KUKA KRL program: MyProgram_103().src

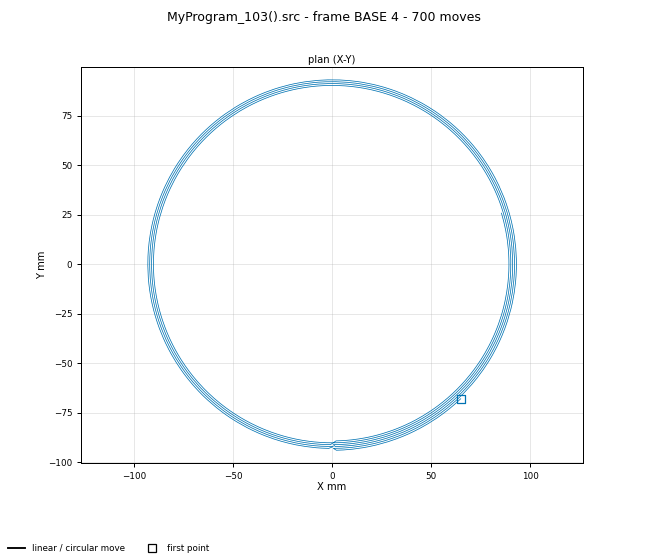
[picture p0: tool path of MyProgram_103().src in frame BASE 4, 700 of 700 moves have a stored position in this frame; points joined in program order, loops and branches not executed]
&ACCESS RVP
&REL 1
&PARAM TEMPLATE = C:\KRC\Roboter\Template\vorgabe
&PARAM EDITMASK = *
DEF MyProgram_103()
; ---- Setting reference (Base) ----
$BASE = BASE_DATA[4]

; --------------------------
; ---- Setting tool (TCP) ----
$TOOL = TOOL_DATA[3]
; --------------------------

$VEL.CP = VEL_APROX_PRINT
Startdeposition()
$VEL.CP = VEL_PRINT
LIN {X 64.9049,Y -67.9874,Z 93,A -51.9833,B 24.9346,C -1.8674,E1 25.1081,E2 497.2894} C_DIS
LIN {X 61.9537,Y -70.6859,Z 93,A -53.7014,B 24.9332,C -1.8881,E1 25.1046,E2 498.9518} C_DIS
LIN {X 59.3764,Y -72.8646,Z 93,A -56.3232,B 24.9349,C -1.863,E1 25.0988,E2 501.6231} C_DIS
LIN {X 56.5767,Y -75.0589,Z 93,A -58.0542,B 24.9341,C -1.8743,E1 25.0951,E2 503.3211} C_DIS
LIN {X 52.9467,Y -77.6626,Z 93,A -60.3598,B 24.9335,C -1.884,E1 25.0899,E2 505.5957} C_DIS
LIN {X 48.6372,Y -80.4313,Z 93,A -63.8521,B 24.9348,C -1.8645,E1 25.0815,E2 509.1227} C_DIS
LIN {X 44.582,Y -82.7481,Z 93,A -66.4916,B 24.9347,C -1.867,E1 25.0752,E2 511.7486} C_DIS
LIN {X 41.1529,Y -84.5065,Z 93,A -68.9502,B 24.9352,C -1.8591,E1 25.069,E2 514.2192} C_DIS
LIN {X 38.4528,Y -85.768,Z 93,A -70.647,B 24.9352,C -1.8607,E1 25.0647,E2 515.908} C_DIS
LIN {X 35.5579,Y -87.008,Z 93,A -72.6876,B 24.9356,C -1.8535,E1 25.0594,E2 517.9607} C_DIS
LIN {X 32.1278,Y -88.332,Z 93,A -74.8746,B 24.9356,C -1.8524,E1 25.0537,E2 520.1456} C_DIS
LIN {X 28.0038,Y -89.7249,Z 93,A -77.5473,B 24.9359,C -1.8485,E1 25.0466,E2 522.8225} C_DIS
LIN {X 22.2186,Y -91.3295,Z 93,A -81.2447,B 24.9363,C -1.8433,E1 25.0366,E2 526.5264} C_DIS
LIN {X 18.4904,Y -92.1576,Z 93,A -83.3808,B 24.936,C -1.848,E1 25.0308,E2 528.6487} C_DIS
LIN {X 15.7341,Y -92.6673,Z 93,A -85.254,B 24.9365,C -1.8409,E1 25.0256,E2 530.5368} C_DIS
LIN {X 10.3903,Y -93.4188,Z 93,A -88.3808,B 24.9362,C -1.8444,E1 25.017,E2 533.6526} C_DIS
LIN {X 5.6146,Y -93.8264,Z 93,A -91.4459,B 24.9367,C -1.838,E1 25.0084,E2 536.7313} C_DIS
LIN {X 2.1765,Y -93.9691,Z 93,A -93.605,B 24.9369,C -1.8351,E1 25.0024,E2 538.8967} C_DIS
LIN {X 2.1765,Y -93.9691,Z 93,A -93.605,B 24.9369,C -1.8351,E1 25.0024,E2 538.8967} C_DIS
Enddeposition()
LIN {X 0.6226,Y -93.0173,Z 93,A -94.0393,B 24.9345,C -1.8697,E1 25.0014,E2 539.2489} C_DIS
Startdeposition()
$VEL.CP = VEL_PRINT
LIN {X 4.8122,Y -92.9245,Z 93,A -89.9697,B 24.9307,C -1.9224,E1 25.0131,E2 535.0555} C_DIS
LIN {X 10.0586,Y -92.5039,Z 93,A -88.0458,B 24.9339,C -1.8776,E1 25.0182,E2 533.2392} C_DIS
LIN {X 16.1981,Y -91.6281,Z 93,A -83.9532,B 24.9331,C -1.8898,E1 25.0295,E2 529.1213} C_DIS
LIN {X 21.4978,Y -90.5327,Z 93,A -80.1723,B 24.9317,C -1.9088,E1 25.0399,E2 525.3004} C_DIS
LIN {X 26.3121,Y -89.2508,Z 93,A -77.5578,B 24.9326,C -1.8959,E1 25.0469,E2 522.7207} C_DIS
LIN {X 29.8863,Y -88.1184,Z 93,A -75.0169,B 24.9318,C -1.9071,E1 25.0537,E2 520.1582} C_DIS
LIN {X 33.849,Y -86.6734,Z 93,A -72.666,B 24.9322,C -1.9017,E1 25.0598,E2 517.8252} C_DIS
LIN {X 36.9367,Y -85.4035,Z 93,A -70.7563,B 24.9324,C -1.8994,E1 25.0647,E2 515.9253} C_DIS
LIN {X 40.1669,Y -83.9324,Z 93,A -67.9542,B 24.9305,C -1.9253,E1 25.0719,E2 513.0693} C_DIS
LIN {X 43.1685,Y -82.429,Z 93,A -66.412,B 24.9316,C -1.9096,E1 25.0756,E2 511.5685} C_DIS
LIN {X 45.3175,Y -81.2671,Z 93,A -64.8499,B 24.9313,C -1.9143,E1 25.0794,E2 509.9997} C_DIS
LIN {X 48.1998,Y -79.5916,Z 93,A -62.4975,B 24.9302,C -1.9291,E1 25.0851,E2 507.6197} C_DIS
LIN {X 52.1558,Y -77.057,Z 93,A -60.0101,B 24.9309,C -1.9198,E1 25.0909,E2 505.1624} C_DIS
LIN {X 55.1018,Y -74.9788,Z 93,A -57.7519,B 24.9305,C -1.9258,E1 25.096,E2 502.898} C_DIS
LIN {X 58.2189,Y -72.5845,Z 93,A -54.9321,B 24.929,C -1.9458,E1 25.1023,E2 500.0413} C_DIS
LIN {X 62.7773,Y -68.6808,Z 93,A -51.4545,B 24.929,C -1.9462,E1 25.1095,E2 496.5767} C_DIS
LIN {X 66.2243,Y -65.3632,Z 93,A -48.3301,B 24.928,C -1.96,E1 25.1157,E2 493.4329} C_DIS
LIN {X 70.519,Y -60.7043,Z 93,A -44.6552,B 24.9279,C -1.9614,E1 25.1226,E2 489.771} C_DIS
LIN {X 73.1256,Y -57.5385,Z 93,A -42.0163,B 24.9271,C -1.9724,E1 25.1272,E2 487.1185} C_DIS
LIN {X 76.178,Y -53.4329,Z 93,A -38.7924,B 24.9262,C -1.9837,E1 25.1325,E2 483.8835} C_DIS
LIN {X 79.1029,Y -48.9987,Z 93,A -35.8993,B 24.9266,C -1.9787,E1 25.1368,E2 481.0166} C_DIS
LIN {X 81.007,Y -45.7832,Z 93,A -32.8346,B 24.9239,C -2.0143,E1 25.1411,E2 477.884} C_DIS
LIN {X 83.1606,Y -41.7437,Z 93,A -30.7888,B 24.9255,C -1.9933,E1 25.1436,E2 475.8985} C_DIS
LIN {X 84.574,Y -38.8009,Z 93,A -28.9541,B 24.9255,C -1.9927,E1 25.1458,E2 474.0751} C_DIS
LIN {X 85.7557,Y -36.1106,Z 93,A -27.0884,B 24.925,C -2.0004,E1 25.1479,E2 472.2015} C_DIS
LIN {X 87.1821,Y -32.5194,Z 93,A -24.5222,B 24.9239,C -2.0147,E1 25.1504,E2 469.6157} C_DIS
LIN {X 88.5131,Y -28.6957,Z 93,A -22.2361,B 24.9239,C -2.0147,E1 25.1525,E2 467.3427} C_DIS
LIN {X 90.2836,Y -22.5193,Z 93,A -18.2449,B 24.9228,C -2.0284,E1 25.1555,E2 463.3419} C_DIS
LIN {X 90.9527,Y -19.638,Z 93,A -15.504,B 24.9197,C -2.0693,E1 25.1571,E2 460.5206} C_DIS
LIN {X 91.9008,Y -14.5732,Z 93,A -13.5998,B 24.9226,C -2.0311,E1 25.1579,E2 458.7176} C_DIS
LIN {X 92.581,Y -9.322,Z 93,A -10.0696,B 24.9211,C -2.0517,E1 25.1592,E2 455.1595} C_DIS
LIN {X 92.8553,Y -5.9982,Z 93,A -7.4727,B 24.9189,C -2.079,E1 25.1596,E2 452.5138} C_DIS
LIN {X 93.0232,Y -2.2255,Z 93,A -5.3762,B 24.919,C -2.0777,E1 25.1598,E2 450.4328} C_DIS
LIN {X 93.0129,Y 2.5845,Z 93,A -2.7784,B 24.9194,C -2.0734,E1 25.1597,E2 447.8605} C_DIS
LIN {X 92.6878,Y 8.1923,Z 93,A 0.3644,B 24.9194,C -2.0725,E1 25.1591,E2 444.7385} C_DIS
LIN {X 91.9596,Y 14.1932,Z 93,A 3.8715,B 24.9192,C -2.0762,E1 25.1579,E2 441.2436} C_DIS
LIN {X 91.3908,Y 17.4854,Z 93,A 6.6018,B 24.9167,C -2.1078,E1 25.1565,E2 438.4545} C_DIS
LIN {X 90.4897,Y 21.671,Z 93,A 9.2019,B 24.9161,C -2.1146,E1 25.1549,E2 435.8536} C_DIS
LIN {X 89.4572,Y 25.6022,Z 93,A 11.8466,B 24.9151,C -2.1275,E1 25.1529,E2 433.1936} C_DIS
LIN {X 87.9202,Y 30.4662,Z 93,A 14.5943,B 24.9155,C -2.1221,E1 25.1505,E2 430.4741} C_DIS
LIN {X 86.7849,Y 33.5653,Z 93,A 16.5323,B 24.9153,C -2.1245,E1 25.1486,E2 428.5413} C_DIS
LIN {X 84.1559,Y 39.6992,Z 93,A 20.551,B 24.9147,C -2.1328,E1 25.1442,E2 424.5249} C_DIS
LIN {X 82.2903,Y 43.4318,Z 93,A 23.7236,B 24.9123,C -2.1624,E1 25.14,E2 421.2993} C_DIS
LIN {X 80.6908,Y 46.3358,Z 93,A 25.2293,B 24.9135,C -2.1479,E1 25.138,E2 419.8355} C_DIS
LIN {X 78.7656,Y 49.5386,Z 93,A 28.4403,B 24.9102,C -2.1878,E1 25.1331,E2 416.5466} C_DIS
LIN {X 76.1381,Y 53.4898,Z 93,A 30.5308,B 24.9121,C -2.1643,E1 25.1299,E2 414.522} C_DIS
LIN {X 73.6324,Y 56.8885,Z 93,A 33.1379,B 24.9116,C -2.1709,E1 25.1255,E2 411.9117} C_DIS
LIN {X 71.2757,Y 59.8163,Z 93,A 35.2495,B 24.9118,C -2.1689,E1 25.1218,E2 409.8147} C_DIS
LIN {X 69.3808,Y 62.0025,Z 93,A 37.7076,B 24.9094,C -2.1977,E1 25.1172,E2 407.2993} C_DIS
LIN {X 66.8807,Y 64.6916,Z 93,A 39.4484,B 24.9106,C -2.1836,E1 25.1139,E2 405.5995} C_DIS
LIN {X 64.3624,Y 67.1981,Z 93,A 41.445,B 24.9108,C -2.1812,E1 25.1099,E2 403.6168} C_DIS
LIN {X 62.0278,Y 69.3582,Z 93,A 43.5422,B 24.91,C -2.1902,E1 25.1055,E2 401.5069} C_DIS
LIN {X 59.3656,Y 71.6503,Z 93,A 45.8089,B 24.9094,C -2.1981,E1 25.1007,E2 399.2303} C_DIS
LIN {X 54.7047,Y 75.2696,Z 93,A 49.3703,B 24.9091,C -2.2019,E1 25.0928,E2 395.6728} C_DIS
LIN {X 51.8989,Y 77.231,Z 93,A 51.6065,B 24.9084,C -2.2099,E1 25.0876,E2 393.425} C_DIS
LIN {X 48.6643,Y 79.3092,Z 93,A 53.9531,B 24.9081,C -2.2128,E1 25.082,E2 391.0791} C_DIS
LIN {X 45.3097,Y 81.2714,Z 93,A 56.5154,B 24.9074,C -2.2222,E1 25.0758,E2 388.5022} C_DIS
LIN {X 39.8165,Y 84.1008,Z 93,A 59.8419,B 24.9084,C -2.21,E1 25.0676,E2 385.2137} C_DIS
LIN {X 35.4139,Y 86.0465,Z 93,A 62.8769,B 24.9079,C -2.2157,E1 25.0598,E2 382.1724} C_DIS
LIN {X 31.8753,Y 87.4184,Z 93,A 65.1162,B 24.908,C -2.2145,E1 25.0539,E2 379.9407} C_DIS
LIN {X 29.3278,Y 88.3067,Z 93,A 66.9704,B 24.9073,C -2.2226,E1 25.049,E2 378.0709} C_DIS
LIN {X 25.9844,Y 89.348,Z 93,A 69.1375,B 24.9072,C -2.2246,E1 25.0432,E2 375.903} C_DIS
LIN {X 22.6331,Y 90.2555,Z 93,A 71.0724,B 24.9076,C -2.2189,E1 25.038,E2 373.9847} C_DIS
LIN {X 20.5715,Y 90.7467,Z 93,A 72.4369,B 24.9074,C -2.2216,E1 25.0343,E2 372.6155} C_DIS
LIN {X 15.3426,Y 91.7748,Z 93,A 75.7008,B 24.9074,C -2.2223,E1 25.0253,E2 369.3537} C_DIS
LIN {X 13.1156,Y 92.1194,Z 93,A 77.9313,B 24.9049,C -2.2518,E1 25.019,E2 367.0552} C_DIS
LIN {X 8.696,Y 92.6413,Z 93,A 79.8432,B 24.9073,C -2.2236,E1 25.0139,E2 365.2115} C_DIS
LIN {X 3.7542,Y 92.973,Z 93,A 82.7917,B 24.9075,C -2.2201,E1 25.0057,E2 362.2724} C_DIS
LIN {X -2.15,Y 93.0246,Z 93,A 86.4724,B 24.9075,C -2.2208,E1 24.9954,E2 358.59} C_DIS
LIN {X -7.3461,Y 92.758,Z 93,A 89.5732,B 24.9079,C -2.2162,E1 24.9868,E2 355.4994} C_DIS
LIN {X -13.9208,Y 92.0017,Z 93,A 94.8926,B 24.9046,C -2.2555,E1 24.9718,E2 350.0827} C_DIS
LIN {X -19.1569,Y 91.0562,Z 93,A 97.185,B 24.9076,C -2.2198,E1 24.9657,E2 347.8725} C_DIS
LIN {X -21.6885,Y 90.4863,Z 93,A 99.0287,B 24.907,C -2.2264,E1 24.9607,E2 346.0105} C_DIS
LIN {X -26.5562,Y 89.1784,Z 93,A 101.8447,B 24.9081,C -2.2137,E1 24.9532,E2 343.2203} C_DIS
LIN {X -29.2761,Y 88.3241,Z 93,A 103.4506,B 24.9087,C -2.2067,E1 24.9489,E2 341.6281} C_DIS
LIN {X -33.6201,Y 86.7634,Z 93,A 106.2312,B 24.9091,C -2.201,E1 24.9417,E2 338.8554} C_DIS
LIN {X -37.1622,Y 85.3052,Z 93,A 108.7868,B 24.9089,C -2.2041,E1 24.935,E2 336.2867} C_DIS
LIN {X -39.1812,Y 84.397,Z 93,A 110.6758,B 24.9076,C -2.2191,E1 24.9302,E2 334.3573} C_DIS
LIN {X -42.1939,Y 82.932,Z 93,A 112.5588,B 24.9084,C -2.2099,E1 24.9255,E2 332.4911} C_DIS
LIN {X -46.113,Y 80.8188,Z 93,A 114.9541,B 24.9097,C -2.1939,E1 24.9197,E2 330.1269} C_DIS
LIN {X -48.8364,Y 79.2042,Z 93,A 116.9522,B 24.9099,C -2.1919,E1 24.915,E2 328.1274} C_DIS
LIN {X -54.2253,Y 75.6153,Z 93,A 120.858,B 24.9107,C -2.1815,E1 24.906,E2 324.2333} C_DIS
LIN {X -55.8386,Y 74.4316,Z 93,A 122.2481,B 24.9105,C -2.184,E1 24.9028,E2 322.8324} C_DIS
LIN {X -58.7964,Y 72.1184,Z 93,A 124.6083,B 24.9108,C -2.1805,E1 24.8977,E2 320.4716} C_DIS
LIN {X -61.4925,Y 69.8343,Z 93,A 126.7951,B 24.9112,C -2.176,E1 24.8931,E2 318.2871} C_DIS
LIN {X -63.8237,Y 67.7093,Z 93,A 128.5532,B 24.912,C -2.1656,E1 24.8895,E2 316.5464} C_DIS
LIN {X -66.0337,Y 65.5562,Z 93,A 130.5936,B 24.912,C -2.1656,E1 24.8854,E2 314.4977} C_DIS
LIN {X -68.3862,Y 63.0984,Z 93,A 132.7073,B 24.9124,C -2.1609,E1 24.8814,E2 312.3858} C_DIS
LIN {X -70.656,Y 60.5459,Z 93,A 134.8199,B 24.9128,C -2.1559,E1 24.8775,E2 310.2757} C_DIS
LIN {X -72.8979,Y 57.8267,Z 93,A 136.9851,B 24.9133,C -2.15,E1 24.8737,E2 308.1143} C_DIS
LIN {X -75.1363,Y 54.8868,Z 93,A 140.1815,B 24.9114,C -2.1729,E1 24.8683,E2 304.8479} C_DIS
LIN {X -77.8782,Y 50.9227,Z 93,A 142.3091,B 24.9143,C -2.1382,E1 24.8651,E2 302.7924} C_DIS
LIN {X -79.6083,Y 48.1721,Z 93,A 143.9836,B 24.9155,C -2.1224,E1 24.8627,E2 301.147} C_DIS
LIN {X -82.0906,Y 43.811,Z 93,A 147.3731,B 24.9155,C -2.1227,E1 24.8581,E2 297.7391} C_DIS
LIN {X -84.4767,Y 39.01,Z 93,A 150.7881,B 24.916,C -2.1164,E1 24.8539,E2 294.3207} C_DIS
LIN {X -85.6745,Y 36.3033,Z 93,A 152.4935,B 24.9167,C -2.1073,E1 24.852,E2 292.6276} C_DIS
LIN {X -86.9887,Y 33.0299,Z 93,A 154.699,B 24.9172,C -2.1017,E1 24.8498,E2 290.4231} C_DIS
LIN {X -88.0749,Y 30.0152,Z 93,A 157.3972,B 24.9159,C -2.1181,E1 24.8473,E2 287.6704} C_DIS
LIN {X -89.2835,Y 26.2021,Z 93,A 159.0869,B 24.9184,C -2.0864,E1 24.846,E2 286.0467} C_DIS
LIN {X -90.2999,Y 22.4524,Z 93,A 161.6573,B 24.9185,C -2.0843,E1 24.8442,E2 283.4662} C_DIS
LIN {X -90.9658,Y 19.5778,Z 93,A 164.1281,B 24.9174,C -2.0988,E1 24.8427,E2 280.9461} C_DIS
LIN {X -91.731,Y 15.6048,Z 93,A 166.068,B 24.9194,C -2.0738,E1 24.8418,E2 279.0546} C_DIS
LIN {X -92.384,Y 11.1033,Z 93,A 168.8022,B 24.9202,C -2.0627,E1 24.8408,E2 276.3304} C_DIS
LIN {X -92.7745,Y 7.1393,Z 93,A 171.7395,B 24.9197,C -2.0699,E1 24.8401,E2 273.3584} C_DIS
LIN {X -92.9725,Y 3.766,Z 93,A 174.1522,B 24.9194,C -2.0736,E1 24.8398,E2 270.9224} C_DIS
LIN {X -93.0461,Y -0.7414,Z 93,A 176.0143,B 24.9223,C -2.0362,E1 24.8398,E2 269.1381} C_DIS
LIN {X -92.7943,Y -6.8918,Z 93,A 179.7782,B 24.9232,C -2.0233,E1 24.8403,E2 265.3826} C_DIS
LIN {X -92.541,Y -9.7046,Z 93,A -178.2438,B 24.9231,C -2.0252,E1 24.8408,E2 263.3881} C_DIS
LIN {X -92.1385,Y -12.9816,Z 93,A -176.2562,B 24.9237,C -2.0174,E1 24.8416,E2 261.4073} C_DIS
LIN {X -91.5803,Y -16.4638,Z 93,A -174.0698,B 24.9242,C -2.011,E1 24.8426,E2 259.2231} C_DIS
LIN {X -90.936,Y -19.7148,Z 93,A -172.0325,B 24.9247,C -2.0046,E1 24.8437,E2 257.189} C_DIS
LIN {X -90.1449,Y -23.0634,Z 93,A -169.8926,B 24.9251,C -1.9988,E1 24.8452,E2 255.0506} C_DIS
LIN {X -89.2609,Y -26.2782,Z 93,A -167.8141,B 24.9255,C -1.9934,E1 24.8468,E2 252.9729} C_DIS
LIN {X -88.2509,Y -29.4934,Z 93,A -165.2425,B 24.9248,C -2.0027,E1 24.849,E2 250.3643} C_DIS
LIN {X -87.1382,Y -32.6352,Z 93,A -163.4778,B 24.9259,C -1.9877,E1 24.8507,E2 248.6256} C_DIS
LIN {X -85.1042,Y -37.6232,Z 93,A -160.2986,B 24.927,C -1.9738,E1 24.8542,E2 245.4618} C_DIS
LIN {X -84.1342,Y -39.7458,Z 93,A -158.7578,B 24.927,C -1.973,E1 24.856,E2 243.9145} C_DIS
LIN {X -82.434,Y -43.1591,Z 93,A -156.5296,B 24.9278,C -1.9628,E1 24.8588,E2 241.6988} C_DIS
LIN {X -81.1903,Y -45.455,Z 93,A -154.5933,B 24.9273,C -1.9688,E1 24.8615,E2 239.7379} C_DIS
LIN {X -78.8229,Y -49.4468,Z 93,A -151.6595,B 24.9277,C -1.9638,E1 24.8658,E2 236.8011} C_DIS
LIN {X -76.3251,Y -53.2213,Z 93,A -149.4062,B 24.9295,C -1.9398,E1 24.8692,E2 234.5939} C_DIS
LIN {X -74.6285,Y -55.5765,Z 93,A -147.4244,B 24.9293,C -1.9415,E1 24.8725,E2 232.5982} C_DIS
LIN {X -72.6469,Y -58.1443,Z 93,A -145.3327,B 24.9295,C -1.9398,E1 24.8761,E2 230.5008} C_DIS
LIN {X -70.1868,Y -61.0889,Z 93,A -142.3863,B 24.9285,C -1.9532,E1 24.8816,E2 227.5091} C_DIS
LIN {X -67.5412,Y -64.0025,Z 93,A -140.5636,B 24.9303,C -1.9285,E1 24.885,E2 225.7373} C_DIS
LIN {X -65.2749,Y -66.3115,Z 93,A -138.5847,B 24.9306,C -1.9239,E1 24.8889,E2 223.7611} C_DIS
LIN {X -62.8649,Y -68.6004,Z 93,A -136.5335,B 24.9309,C -1.9199,E1 24.8931,E2 221.711} C_DIS
LIN {X -58.3134,Y -72.5087,Z 93,A -132.3061,B 24.9301,C -1.9303,E1 24.9022,E2 217.4425} C_DIS
LIN {X -55.4939,Y -74.6905,Z 93,A -130.7772,B 24.932,C -1.9046,E1 24.9055,E2 215.9694} C_DIS
LIN {X -53.5385,Y -76.1046,Z 93,A -129.06,B 24.9316,C -1.9097,E1 24.9094,E2 214.2341} C_DIS
LIN {X -51.3498,Y -77.5966,Z 93,A -127.2917,B 24.9315,C -1.9116,E1 24.9136,E2 212.4553} C_DIS
LIN {X -48.2652,Y -79.5518,Z 93,A -125.0341,B 24.9317,C -1.9086,E1 24.9189,E2 210.198} C_DIS
LIN {X -43.0497,Y -82.4915,Z 93,A -121.5436,B 24.9325,C -1.8971,E1 24.9275,E2 206.7249} C_DIS
LIN {X -40.4293,Y -83.8063,Z 93,A -119.4818,B 24.9321,C -1.9035,E1 24.9327,E2 204.6425} C_DIS
LIN {X -37.0801,Y -85.341,Z 93,A -117.2952,B 24.9324,C -1.8982,E1 24.9382,E2 202.4631} C_DIS
LIN {X -33.9612,Y -86.6294,Z 93,A -115.4811,B 24.9332,C -1.8874,E1 24.9429,E2 200.6708} C_DIS
LIN {X -29.3661,Y -88.2938,Z 93,A -112.3109,B 24.933,C -1.8902,E1 24.9513,E2 197.4877} C_DIS
LIN {X -25.9229,Y -89.3663,Z 93,A -110.1905,B 24.9334,C -1.8852,E1 24.9569,E2 195.3756} C_DIS
LIN {X -21.9573,Y -90.4207,Z 93,A -106.9754,B 24.9318,C -1.9073,E1 24.9658,E2 192.1033} C_DIS
LIN {X -18.1137,Y -91.2698,Z 93,A -105.1181,B 24.9333,C -1.8868,E1 24.9707,E2 190.2926} C_DIS
LIN {X -13.4599,Y -92.0702,Z 93,A -102.2849,B 24.9335,C -1.8834,E1 24.9785,E2 187.4648} C_DIS
LIN {X -8.0955,Y -92.6967,Z 93,A -98.8849,B 24.9333,C -1.8856,E1 24.988,E2 184.0577} C_DIS
LIN {X -5.202,Y -92.9029,Z 93,A -96.6288,B 24.9322,C -1.902,E1 24.9944,E2 181.7618} C_DIS
LIN {X -1.696,Y -93.033,Z 93,A -94.144,B 24.9313,C -1.9139,E1 25.0014,E2 179.2489} C_DIS
LIN {X -1.696,Y -93.033,Z 93,A -94.144,B 24.9313,C -1.9139,E1 25.0014,E2 179.2489} C_DIS
Enddeposition()
LIN {X 0.6186,Y -92.0937,Z 93,A -94.2011,B 24.9338,C -1.8791,E1 25.001,E2 179.3884} C_DIS
Startdeposition()
$VEL.CP = VEL_PRINT
LIN {X -5.5387,Y -91.938,Z 93,A -98.1986,B 24.9343,C -1.8728,E1 24.9898,E2 183.4015} C_DIS
LIN {X -8.9285,Y -91.67,Z 93,A -100.6468,B 24.935,C -1.8618,E1 24.9829,E2 185.877} C_DIS
LIN {X -11.5193,Y -91.3809,Z 93,A -102.7076,B 24.936,C -1.8475,E1 24.9771,E2 187.9733} C_DIS
LIN {X -15.144,Y -90.85,Z 93,A -104.3705,B 24.9346,C -1.8685,E1 24.9727,E2 189.5878} C_DIS
LIN {X -18.596,Y -90.2068,Z 93,A -106.9037,B 24.9353,C -1.8578,E1 24.9657,E2 192.1491} C_DIS
LIN {X -23.3964,Y -89.0837,Z 93,A -109.5092,B 24.9341,C -1.8747,E1 24.9587,E2 194.7183} C_DIS
LIN {X -26.3206,Y -88.2627,Z 93,A -111.6035,B 24.9345,C -1.8692,E1 24.953,E2 196.8289} C_DIS
LIN {X -29.7496,Y -87.1673,Z 93,A -114.3672,B 24.9356,C -1.854,E1 24.9456,E2 199.634} C_DIS
LIN {X -33.2061,Y -85.9109,Z 93,A -115.8986,B 24.9337,C -1.8806,E1 24.9418,E2 201.1054} C_DIS
LIN {X -36.9723,Y -84.3573,Z 93,A -118.645,B 24.934,C -1.8763,E1 24.9346,E2 203.8682} C_DIS
LIN {X -40.3598,Y -82.7915,Z 93,A -121.0579,B 24.934,C -1.8761,E1 24.9285,E2 206.2878} C_DIS
LIN {X -43.4794,Y -81.1964,Z 93,A -123.9809,B 24.9355,C -1.8552,E1 24.9212,E2 209.2685} C_DIS
LIN {X -47.4405,Y -78.9473,Z 93,A -125.7955,B 24.9329,C -1.8917,E1 24.917,E2 211.0019} C_DIS
LIN {X -50.0737,Y -77.3035,Z 93,A -127.8134,B 24.9329,C -1.8918,E1 24.9122,E2 213.0259} C_DIS
LIN {X -51.8344,Y -76.1336,Z 93,A -129.4133,B 24.9334,C -1.8849,E1 24.9085,E2 214.6476} C_DIS
LIN {X -54.8121,Y -74.0199,Z 93,A -132.4895,B 24.9349,C -1.8636,E1 24.9015,E2 217.7854} C_DIS
LIN {X -58.7167,Y -70.961,Z 93,A -134.9519,B 24.9331,C -1.8887,E1 24.8962,E2 220.1973} C_DIS
LIN {X -61.4744,Y -68.5855,Z 93,A -136.8393,B 24.932,C -1.9049,E1 24.8924,E2 222.0535} C_DIS
LIN {X -64.1598,Y -66.081,Z 93,A -139.2401,B 24.9319,C -1.906,E1 24.8875,E2 224.4618} C_DIS
LIN {X -66.5497,Y -63.6736,Z 93,A -141.4489,B 24.9318,C -1.9074,E1 24.8832,E2 226.6766} C_DIS
LIN {X -70.3145,Y -59.4898,Z 93,A -144.7094,B 24.9307,C -1.9228,E1 24.8772,E2 229.9151} C_DIS
LIN {X -72.2382,Y -57.1376,Z 93,A -146.6739,B 24.9305,C -1.9249,E1 24.8737,E2 231.8837} C_DIS
LIN {X -74.5899,Y -54.0336,Z 93,A -148.9713,B 24.9298,C -1.9347,E1 24.8699,E2 234.1689} C_DIS
LIN {X -75.983,Y -52.0568,Z 93,A -150.6275,B 24.9298,C -1.9338,E1 24.8672,E2 235.8355} C_DIS
LIN {X -78.6634,Y -47.9076,Z 93,A -153.5177,B 24.9289,C -1.9473,E1 24.8629,E2 238.708} C_DIS
LIN {X -80.498,Y -44.7567,Z 93,A -156.0919,B 24.9291,C -1.944,E1 24.8593,E2 241.3035} C_DIS
LIN {X -82.1839,Y -41.5814,Z 93,A -158.4553,B 24.929,C -1.9463,E1 24.8563,E2 243.6742} C_DIS
LIN {X -83.8835,Y -38.0351,Z 93,A -160.7552,B 24.9282,C -1.9576,E1 24.8536,E2 245.9596} C_DIS
LIN {X -86.0828,Y -32.7541,Z 93,A -165.0978,B 24.9291,C -1.9444,E1 24.849,E2 250.358} C_DIS
LIN {X -87.5142,Y -28.7136,Z 93,A -166.9227,B 24.9267,C -1.9775,E1 24.8475,E2 252.1143} C_DIS
LIN {X -88.3928,Y -25.8823,Z 93,A -168.9612,B 24.9267,C -1.9772,E1 24.8458,E2 254.1653} C_DIS
LIN {X -89.3176,Y -22.4867,Z 93,A -171.0569,B 24.926,C -1.9866,E1 24.8443,E2 256.2506} C_DIS
LIN {X -90.0351,Y -19.4111,Z 93,A -173.1392,B 24.9258,C -1.9892,E1 24.8431,E2 258.3391} C_DIS
LIN {X -90.7504,Y -15.7397,Z 93,A -175.509,B 24.9254,C -1.9951,E1 24.8419,E2 260.7088} C_DIS
LIN {X -91.3109,Y -12.06,Z 93,A -177.7444,B 24.9246,C -2.0048,E1 24.841,E2 262.9344} C_DIS
LIN {X -91.7956,Y -7.5275,Z 93,A 179.6435,B 24.9235,C -2.0205,E1 24.8403,E2 265.5248} C_DIS
LIN {X -92.0602,Y -2.8261,Z 93,A 176.5948,B 24.923,C -2.0262,E1 24.8398,E2 268.5781} C_DIS
LIN {X -92.1061,Y 0.0717,Z 93,A 174.0511,B 24.9243,C -2.0099,E1 24.8398,E2 271.1761} C_DIS
LIN {X -92.0319,Y 3.6462,Z 93,A 172.1283,B 24.923,C -2.026,E1 24.84,E2 273.072} C_DIS
LIN {X -91.7732,Y 7.8081,Z 93,A 169.7509,B 24.9219,C -2.0408,E1 24.8405,E2 275.4285} C_DIS
LIN {X -91.436,Y 11.0756,Z 93,A 167.7939,B 24.9212,C -2.0499,E1 24.8411,E2 277.3754} C_DIS
LIN {X -90.7504,Y 15.7399,Z 93,A 164.3232,B 24.9217,C -2.0433,E1 24.8426,E2 280.8826} C_DIS
LIN {X -89.6662,Y 21.0511,Z 93,A 161.325,B 24.92,C -2.0651,E1 24.8444,E2 283.8464} C_DIS
LIN {X -88.5781,Y 25.2392,Z 93,A 158.858,B 24.9188,C -2.0803,E1 24.8462,E2 286.2914} C_DIS
LIN {X -87.1392,Y 29.833,Z 93,A 155.9079,B 24.918,C -2.0909,E1 24.8487,E2 289.2331} C_DIS
LIN {X -85.4687,Y 34.3272,Z 93,A 152.7175,B 24.9178,C -2.0938,E1 24.8518,E2 292.4345} C_DIS
LIN {X -84.1883,Y 37.3588,Z 93,A 150.5728,B 24.9175,C -2.0971,E1 24.8542,E2 294.5833} C_DIS
LIN {X -81.7577,Y 42.4135,Z 93,A 147.2847,B 24.9162,C -2.1134,E1 24.8582,E2 297.8501} C_DIS
LIN {X -80.5485,Y 44.6659,Z 93,A 145.0797,B 24.9173,C -2.0996,E1 24.8612,E2 300.0996} C_DIS
LIN {X -78.0016,Y 48.9782,Z 93,A 141.5534,B 24.9176,C -2.0962,E1 24.8665,E2 303.6522} C_DIS
LIN {X -75.6071,Y 52.5985,Z 93,A 139.4441,B 24.9156,C -2.1213,E1 24.8697,E2 305.712} C_DIS
LIN {X -73.5694,Y 55.4133,Z 93,A 137.3948,B 24.9149,C -2.1305,E1 24.8731,E2 307.7492} C_DIS
LIN {X -71.4117,Y 58.1677,Z 93,A 135.2118,B 24.9144,C -2.136,E1 24.8769,E2 309.9293} C_DIS
LIN {X -69.1491,Y 60.8406,Z 93,A 133.0005,B 24.9141,C -2.1406,E1 24.8809,E2 312.1398} C_DIS
LIN {X -66.7344,Y 63.4812,Z 93,A 130.7442,B 24.9137,C -2.1452,E1 24.8852,E2 314.3951} C_DIS
LIN {X -64.2446,Y 65.9993,Z 93,A 128.6988,B 24.9129,C -2.1553,E1 24.8892,E2 316.425} C_DIS
LIN {X -62.2101,Y 67.9189,Z 93,A 126.9403,B 24.9126,C -2.1588,E1 24.8928,E2 318.1823} C_DIS
LIN {X -59.793,Y 70.0562,Z 93,A 124.8642,B 24.9124,C -2.1612,E1 24.8972,E2 320.2609} C_DIS
LIN {X -56.7107,Y 72.5756,Z 93,A 122.2466,B 24.9124,C -2.1621,E1 24.9029,E2 322.8859} C_DIS
LIN {X -54.1338,Y 74.5166,Z 93,A 120.2576,B 24.9119,C -2.1668,E1 24.9074,E2 324.8707} C_DIS
LIN {X -48.6077,Y 78.233,Z 93,A 116.5089,B 24.9103,C -2.1871,E1 24.916,E2 328.5836} C_DIS
LIN {X -46.7023,Y 79.3851,Z 93,A 114.7321,B 24.9111,C -2.1774,E1 24.9204,E2 330.389} C_DIS
LIN {X -42.0405,Y 81.9493,Z 93,A 111.7338,B 24.9098,C -2.1927,E1 24.9277,E2 333.3591} C_DIS
LIN {X -39.9321,Y 82.997,Z 93,A 110.0957,B 24.9101,C -2.1896,E1 24.9318,E2 335.009} C_DIS
LIN {X -36.9671,Y 84.3595,Z 93,A 107.9569,B 24.9101,C -2.1892,E1 24.9373,E2 337.154} C_DIS
LIN {X -32.5158,Y 86.1731,Z 93,A 104.4195,B 24.9112,C -2.176,E1 24.9466,E2 340.7303} C_DIS
LIN {X -29.1709,Y 87.3625,Z 93,A 102.9983,B 24.9089,C -2.2036,E1 24.9502,E2 342.0885} C_DIS
LIN {X -26.9036,Y 88.0876,Z 93,A 101.2086,B 24.9096,C -2.1954,E1 24.955,E2 343.9009} C_DIS
LIN {X -23.1368,Y 89.1505,Z 93,A 98.9549,B 24.9089,C -2.2038,E1 24.961,E2 346.1383} C_DIS
LIN {X -20.2989,Y 89.84,Z 93,A 96.9357,B 24.9093,C -2.1989,E1 24.9665,E2 348.1716} C_DIS
LIN {X -14.7085,Y 90.9229,Z 93,A 93.6417,B 24.9084,C -2.2097,E1 24.9755,E2 351.4436} C_DIS
LIN {X -9.7778,Y 91.5833,Z 93,A 90.3986,B 24.9087,C -2.2067,E1 24.9845,E2 354.6961} C_DIS
LIN {X -6.8158,Y 91.8525,Z 93,A 87.8817,B 24.9104,C -2.1859,E1 24.9917,E2 357.2635} C_DIS
LIN {X -3.0709,Y 92.0527,Z 93,A 86.3581,B 24.9081,C -2.213,E1 24.9957,E2 358.723} C_DIS
LIN {X 1.9578,Y 92.0831,Z 93,A 83.2293,B 24.9081,C -2.2136,E1 25.0045,E2 361.8503} C_DIS
LIN {X 7.7838,Y 91.7752,Z 93,A 79.5899,B 24.9081,C -2.2132,E1 25.0146,E2 365.4891} C_DIS
LIN {X 11.9993,Y 91.3187,Z 93,A 77.1377,B 24.9076,C -2.219,E1 25.0214,E2 367.9259} C_DIS
LIN {X 14.0983,Y 91.0182,Z 93,A 75.5199,B 24.9085,C -2.2086,E1 25.0259,E2 369.5668} C_DIS
LIN {X 20.2234,Y 89.8574,Z 93,A 71.7551,B 24.9083,C -2.2107,E1 25.0362,E2 373.3221} C_DIS
LIN {X 23.6825,Y 89.0075,Z 93,A 69.324,B 24.909,C -2.2022,E1 25.0428,E2 375.7699} C_DIS
LIN {X 27.0735,Y 88.0349,Z 93,A 67.0926,B 24.9093,C -2.1993,E1 25.0488,E2 378.0041} C_DIS
LIN {X 30.5364,Y 86.8942,Z 93,A 64.9037,B 24.9093,C -2.2001,E1 25.0546,E2 380.1869} C_DIS
LIN {X 34.0914,Y 85.5631,Z 93,A 62.3566,B 24.9099,C -2.1915,E1 25.0612,E2 382.7489} C_DIS
LIN {X 37.3491,Y 84.1926,Z 93,A 60.3596,B 24.9095,C -2.196,E1 25.0663,E2 384.7305} C_DIS
LIN {X 40.2618,Y 82.8386,Z 93,A 57.5337,B 24.9121,C -2.1653,E1 25.0736,E2 387.6216} C_DIS
LIN {X 44.3126,Y 80.7445,Z 93,A 55.684,B 24.9096,C -2.1953,E1 25.078,E2 389.3949} C_DIS
LIN {X 47.0122,Y 79.202,Z 93,A 53.6248,B 24.9102,C -2.1882,E1 25.083,E2 391.4646} C_DIS
LIN {X 50.3984,Y 77.0916,Z 93,A 51.3062,B 24.91,C -2.1901,E1 25.0884,E2 393.7714} C_DIS
LIN {X 52.4482,Y 75.7118,Z 93,A 49.6493,B 24.9106,C -2.1833,E1 25.0922,E2 395.4386} C_DIS
LIN {X 55.1586,Y 73.7607,Z 93,A 46.7552,B 24.9132,C -2.1513,E1 25.0989,E2 398.398} C_DIS
LIN {X 58.6084,Y 71.051,Z 93,A 44.9474,B 24.911,C -2.1784,E1 25.1027,E2 400.1351} C_DIS
LIN {X 60.6932,Y 69.2779,Z 93,A 43.0811,B 24.9117,C -2.1693,E1 25.1066,E2 402.0155} C_DIS
LIN {X 63.2134,Y 66.9863,Z 93,A 41.0087,B 24.912,C -2.1666,E1 25.1109,E2 404.0858} C_DIS
LIN {X 65.6589,Y 64.5911,Z 93,A 38.8189,B 24.9125,C -2.16,E1 25.1152,E2 406.2821} C_DIS
LIN {X 69.7067,Y 60.2023,Z 93,A 35.3536,B 24.9125,C -2.1605,E1 25.1217,E2 409.7308} C_DIS
LIN {X 71.3735,Y 58.2149,Z 93,A 33.2278,B 24.9142,C -2.1385,E1 25.1255,E2 411.8988} C_DIS
LIN {X 73.6674,Y 55.2827,Z 93,A 31.2907,B 24.9136,C -2.1464,E1 25.1287,E2 413.8081} C_DIS
LIN {X 75.9886,Y 52.0466,Z 93,A 28.3713,B 24.9154,C -2.1243,E1 25.1335,E2 416.7652} C_DIS
LIN {X 77.81,Y 49.2847,Z 93,A 26.9278,B 24.914,C -2.141,E1 25.1356,E2 418.1621} C_DIS
LIN {X 79.0101,Y 47.3368,Z 93,A 25.2888,B 24.915,C -2.1295,E1 25.138,E2 419.8198} C_DIS
LIN {X 82.6146,Y 40.7178,Z 93,A 20.9401,B 24.915,C -2.129,E1 25.1437,E2 424.147} C_DIS
LIN {X 83.6136,Y 38.6246,Z 93,A 18.4457,B 24.9183,C -2.087,E1 25.1467,E2 426.727} C_DIS
LIN {X 85.4116,Y 34.4675,Z 93,A 16.5264,B 24.9164,C -2.1112,E1 25.1487,E2 428.5785} C_DIS
LIN {X 86.6235,Y 31.2972,Z 93,A 14.3386,B 24.9171,C -2.1023,E1 25.1508,E2 430.7753} C_DIS
LIN {X 88.2466,Y 26.3752,Z 93,A 11.1882,B 24.9177,C -2.0953,E1 25.1535,E2 433.9242} C_DIS
LIN {X 89.1749,Y 23.0417,Z 93,A 8.6501,B 24.9193,C -2.0747,E1 25.1553,E2 436.4963} C_DIS
LIN {X 90.6798,Y 16.1331,Z 93,A 4.8963,B 24.9185,C -2.0846,E1 25.1575,E2 440.2048} C_DIS
LIN {X 91.081,Y 13.6921,Z 93,A 2.5751,B 24.9211,C -2.0512,E1 25.1584,E2 442.5912} C_DIS
LIN {X 91.5437,Y 10.1456,Z 93,A 0.8823,B 24.9201,C -2.0636,E1 25.159,E2 444.2448} C_DIS
LIN {X 92.0445,Y 3.3391,Z 93,A -3.3442,B 24.9211,C -2.0507,E1 25.1597,E2 448.4766} C_DIS
LIN {X 92.1003,Y -0.8181,Z 93,A -5.8967,B 24.9217,C -2.0437,E1 25.1597,E2 451.0304} C_DIS
LIN {X 91.9784,Y -4.785,Z 93,A -8.6566,B 24.9231,C -2.0251,E1 25.1594,E2 453.8178} C_DIS
LIN {X 91.7419,Y -8.1603,Z 93,A -11.6973,B 24.9262,C -1.9843,E1 25.1587,E2 456.9366} C_DIS
LIN {X 90.9933,Y -14.2593,Z 93,A -14.5857,B 24.9246,C -2.0059,E1 25.1575,E2 459.7572} C_DIS
LIN {X 89.8895,Y -20.0788,Z 93,A -17.6799,B 24.9238,C -2.0159,E1 25.1558,E2 462.8099} C_DIS
LIN {X 88.8958,Y -24.0959,Z 93,A -20.9155,B 24.9262,C -1.9835,E1 25.1535,E2 466.1032} C_DIS
LIN {X 87.9515,Y -27.3425,Z 93,A -22.39,B 24.925,C -1.9999,E1 25.1523,E2 467.5306} C_DIS
LIN {X 86.9979,Y -30.2408,Z 93,A -24.7483,B 24.9267,C -1.9771,E1 25.1501,E2 469.9293} C_DIS
LIN {X 85.4433,Y -34.3896,Z 93,A -27.5237,B 24.9274,C -1.968,E1 25.1473,E2 472.7109} C_DIS
LIN {X 83.8395,Y -38.1327,Z 93,A -29.6442,B 24.9268,C -1.9754,E1 25.1449,E2 474.8024} C_DIS
LIN {X 81.4905,Y -42.9227,Z 93,A -33.1888,B 24.9282,C -1.9573,E1 25.1405,E2 478.3708} C_DIS
LIN {X 80.0303,Y -45.5889,Z 93,A -34.8885,B 24.9281,C -1.9587,E1 25.1382,E2 480.0582} C_DIS
LIN {X 78.1444,Y -48.7497,Z 93,A -37.6901,B 24.9299,C -1.9336,E1 25.134,E2 482.9048} C_DIS
LIN {X 76.1084,Y -51.8716,Z 93,A -39.2063,B 24.9282,C -1.9563,E1 25.1317,E2 484.3601} C_DIS
LIN {X 74.7613,Y -53.7955,Z 93,A -40.9106,B 24.9292,C -1.9434,E1 25.1289,E2 486.0865} C_DIS
LIN {X 71.6546,Y -57.8681,Z 93,A -44.7268,B 24.9314,C -1.9122,E1 25.1222,E2 489.9585} C_DIS
LIN {X 68.9723,Y -61.0423,Z 93,A -46.4246,B 24.9296,C -1.9375,E1 25.1193,E2 491.5888} C_DIS
LIN {X 67.125,Y -63.0659,Z 93,A -48.9762,B 24.9321,C -1.9028,E1 25.1142,E2 494.2112} C_DIS
LIN {X 64.2635,Y -65.9809,Z 93,A -51.4934,B 24.9325,C -1.8975,E1 25.1092,E2 496.7304} C_DIS
LIN {X 61.3736,Y -68.6758,Z 93,A -53.0729,B 24.9307,C -1.9233,E1 25.1061,E2 498.2427} C_DIS
LIN {X 59.3403,Y -70.4419,Z 93,A -55.6316,B 24.9332,C -1.8879,E1 25.1005,E2 500.8751} C_DIS
LIN {X 56.2071,Y -72.9646,Z 93,A -57.7481,B 24.9326,C -1.8963,E1 25.0959,E2 502.964} C_DIS
LIN {X 53.3432,Y -75.084,Z 93,A -59.7023,B 24.9323,C -1.901,E1 25.0915,E2 504.9001} C_DIS
LIN {X 50.5466,Y -76.9944,Z 93,A -61.6411,B 24.9321,C -1.9028,E1 25.087,E2 506.8281} C_DIS
LIN {X 47.2005,Y -79.0906,Z 93,A -64.6072,B 24.9337,C -1.8802,E1 25.0798,E2 509.8385} C_DIS
LIN {X 44.4159,Y -80.6884,Z 93,A -66.0121,B 24.9325,C -1.8976,E1 25.0765,E2 511.1981} C_DIS
LIN {X 42.2116,Y -81.8618,Z 93,A -67.8755,B 24.9335,C -1.884,E1 25.0718,E2 513.0884} C_DIS
LIN {X 39.1777,Y -83.3564,Z 93,A -70.2647,B 24.9344,C -1.8707,E1 25.0657,E2 515.503} C_DIS
LIN {X 36.1932,Y -84.6955,Z 93,A -71.6272,B 24.933,C -1.8912,E1 25.0624,E2 516.8137} C_DIS
LIN {X 30.8803,Y -86.7723,Z 93,A -75.4878,B 24.9341,C -1.8754,E1 25.0522,E2 520.7031} C_DIS
LIN {X 27.6531,Y -87.8552,Z 93,A -77.4837,B 24.9339,C -1.8771,E1 25.047,E2 522.6914} C_DIS
LIN {X 24.5093,Y -88.7841,Z 93,A -80.0177,B 24.9353,C -1.8578,E1 25.04,E2 525.267} C_DIS
LIN {X 21.2343,Y -89.6239,Z 93,A -82.0707,B 24.9353,C -1.8574,E1 25.0345,E2 527.3178} C_DIS
LIN {X 16.6351,Y -90.5895,Z 93,A -85.7444,B 24.9373,C -1.8296,E1 25.0242,E2 531.0532} C_DIS
LIN {X 10.8743,Y -91.4595,Z 93,A -89.3407,B 24.9373,C -1.8284,E1 25.0142,E2 534.6498} C_DIS
LIN {X 5.1415,Y -91.96,Z 93,A -91.2923,B 24.9336,C -1.8818,E1 25.0092,E2 536.474} C_DIS
LIN {X 1.6208,Y -92.0893,Z 93,A -94.1518,B 24.9353,C -1.8583,E1 25.001,E2 539.3884} C_DIS
LIN {X 1.6208,Y -92.0893,Z 93,A -94.1518,B 24.9353,C -1.8583,E1 25.001,E2 539.3884} C_DIS
Enddeposition()
LIN {X 0.5953,Y -91.1533,Z 93,A -93.149,B 24.9301,C -1.9305,E1 25.0043,E2 538.2146} C_DIS
Startdeposition()
$VEL.CP = VEL_PRINT
LIN {X 4.1257,Y -91.0656,Z 93,A -91.3962,B 24.9312,C -1.9152,E1 25.0091,E2 536.4986} C_DIS
LIN {X 7.0295,Y -90.8876,Z 93,A -88.9283,B 24.9296,C -1.9381,E1 25.0161,E2 533.9776} C_DIS
LIN {X 10.9739,Y -90.4966,Z 93,A -87.2605,B 24.9315,C -1.9111,E1 25.0206,E2 532.375} C_DIS
LIN {X 15.9429,Y -89.754,Z 93,A -83.9577,B 24.931,C -1.9184,E1 25.0297,E2 529.0582} C_DIS
LIN {X 19.4059,Y -89.0692,Z 93,A -81.7903,B 24.931,C -1.9185,E1 25.0356,E2 526.8931} C_DIS
LIN {X 21.7921,Y -88.5158,Z 93,A -79.5548,B 24.9291,C -1.9444,E1 25.0418,E2 524.5995} C_DIS
LIN {X 25.5648,Y -87.5014,Z 93,A -77.7281,B 24.9305,C -1.925,E1 25.0466,E2 522.8219} C_DIS
LIN {X 28.7501,Y -86.5072,Z 93,A -75.909,B 24.931,C -1.9178,E1 25.0514,E2 521.0233} C_DIS
LIN {X 34.4323,Y -84.4058,Z 93,A -71.9025,B 24.9302,C -1.9298,E1 25.0619,E2 516.9968} C_DIS
LIN {X 38.9679,Y -82.4119,Z 93,A -68.674,B 24.9295,C -1.9386,E1 25.0702,E2 513.7556} C_DIS
LIN {X 43.0607,Y -80.3486,Z 93,A -65.9074,B 24.9295,C -1.9394,E1 25.077,E2 510.9949} C_DIS
LIN {X 46.1958,Y -78.587,Z 93,A -63.5899,B 24.929,C -1.9455,E1 25.0826,E2 508.6698} C_DIS
LIN {X 49.676,Y -76.4361,Z 93,A -61.174,B 24.929,C -1.9448,E1 25.0883,E2 506.2633} C_DIS
LIN {X 52.0543,Y -74.8349,Z 93,A -59.2253,B 24.9284,C -1.9537,E1 25.0928,E2 504.3002} C_DIS
LIN {X 54.3995,Y -73.1492,Z 93,A -57.3826,B 24.9281,C -1.9585,E1 25.097,E2 502.4529} C_DIS
LIN {X 58.1218,Y -70.2268,Z 93,A -54.5284,B 24.9279,C -1.9606,E1 25.1032,E2 499.6043} C_DIS
LIN {X 60.7008,Y -68.0099,Z 93,A -52.4271,B 24.9277,C -1.9642,E1 25.1076,E2 497.5027} C_DIS
LIN {X 64.0341,Y -64.881,Z 93,A -49.198,B 24.9262,C -1.984,E1 25.1142,E2 494.2403} C_DIS
LIN {X 67.2267,Y -61.567,Z 93,A -46.6714,B 24.9267,C -1.9779,E1 25.119,E2 491.7392} C_DIS
LIN {X 69.4368,Y -59.0631,Z 93,A -44.2325,B 24.9253,C -1.9957,E1 25.1235,E2 489.2693} C_DIS
LIN {X 72.717,Y -54.9749,Z 93,A -41.2665,B 24.9256,C -1.9924,E1 25.1285,E2 486.325} C_DIS
LIN {X 74.6431,Y -52.3302,Z 93,A -39.1733,B 24.925,C -1.9994,E1 25.1319,E2 484.2255} C_DIS
LIN {X 76.0374,Y -50.2816,Z 93,A -37.3585,B 24.924,C -2.0132,E1 25.1348,E2 482.387} C_DIS
LIN {X 78.4883,Y -46.3628,Z 93,A -34.8079,B 24.9244,C -2.0085,E1 25.1384,E2 479.8607} C_DIS
LIN {X 79.5595,Y -44.4994,Z 93,A -32.1363,B 24.9203,C -2.0615,E1 25.1422,E2 477.0779} C_DIS
LIN {X 82.44,Y -38.9074,Z 93,A -29.4943,B 24.9232,C -2.0244,E1 25.1453,E2 474.5376} C_DIS
LIN {X 84.4714,Y -34.2712,Z 93,A -26.5071,B 24.923,C -2.0269,E1 25.1485,E2 471.5609} C_DIS
LIN {X 86.1229,Y -29.8809,Z 93,A -23.3823,B 24.9218,C -2.0425,E1 25.1515,E2 468.4168} C_DIS
LIN {X 87.2167,Y -26.522,Z 93,A -20.413,B 24.9191,C -2.0773,E1 25.154,E2 465.3822} C_DIS
LIN {X 88.4283,Y -22.1506,Z 93,A -18.3694,B 24.9207,C -2.0562,E1 25.1554,E2 463.4001} C_DIS
LIN {X 89.2589,Y -18.5146,Z 93,A -15.393,B 24.9183,C -2.0872,E1 25.1572,E2 460.368} C_DIS
LIN {X 90.0034,Y -14.4777,Z 93,A -13.6696,B 24.9201,C -2.0636,E1 25.1579,E2 458.7103} C_DIS
LIN {X 90.7327,Y -8.814,Z 93,A -9.9516,B 24.9189,C -2.0798,E1 25.1592,E2 454.976} C_DIS
LIN {X 90.9709,Y -5.8562,Z 93,A -7.7055,B 24.9173,C -2.1,E1 25.1596,E2 452.6957} C_DIS
LIN {X 91.1213,Y -2.6168,Z 93,A -5.1818,B 24.9153,C -2.1247,E1 25.1598,E2 450.1287} C_DIS
LIN {X 91.1338,Y 2.1909,Z 93,A -2.7047,B 24.9162,C -2.114,E1 25.1597,E2 447.6916} C_DIS
LIN {X 90.7625,Y 8.4908,Z 93,A 0.4457,B 24.9176,C -2.0965,E1 25.1591,E2 444.6011} C_DIS
LIN {X 90.2445,Y 12.878,Z 93,A 3.5547,B 24.9159,C -2.1174,E1 25.158,E2 441.4611} C_DIS
LIN {X 89.7399,Y 16.0213,Z 93,A 5.5667,B 24.9154,C -2.1241,E1 25.1571,E2 439.4452} C_DIS
LIN {X 88.8776,Y 20.2669,Z 93,A 8.4265,B 24.9143,C -2.1375,E1 25.1554,E2 436.5704} C_DIS
LIN {X 87.8823,Y 24.2248,Z 93,A 10.8554,B 24.9141,C -2.1403,E1 25.1537,E2 434.1488} C_DIS
LIN {X 87.0962,Y 26.9105,Z 93,A 12.8434,B 24.913,C -2.1541,E1 25.152,E2 432.1397} C_DIS
LIN {X 85.7015,Y 31.0675,Z 93,A 15.3875,B 24.913,C -2.1544,E1 25.1497,E2 429.6091} C_DIS
LIN {X 84.5071,Y 34.1835,Z 93,A 17.7507,B 24.9117,C -2.1703,E1 25.1472,E2 427.2216} C_DIS
LIN {X 82.3768,Y 39.0412,Z 93,A 20.7936,B 24.9117,C -2.169,E1 25.1437,E2 424.198} C_DIS
LIN {X 81.0008,Y 41.8201,Z 93,A 23.3696,B 24.9094,C -2.1974,E1 25.1404,E2 421.5688} C_DIS
LIN {X 79.087,Y 45.334,Z 93,A 25.1713,B 24.911,C -2.1781,E1 25.138,E2 419.8219} C_DIS
LIN {X 77.6375,Y 47.7765,Z 93,A 26.9438,B 24.9107,C -2.1823,E1 25.1354,E2 418.0486} C_DIS
LIN {X 75.8372,Y 50.585,Z 93,A 29.3995,B 24.9092,C -2.2007,E1 25.1316,E2 415.5616} C_DIS
LIN {X 73.1509,Y 54.3972,Z 93,A 31.978,B 24.9096,C -2.1952,E1 25.1274,E2 413.0087} C_DIS
LIN {X 71.6085,Y 56.4106,Z 93,A 33.6512,B 24.9091,C -2.2019,E1 25.1245,E2 411.3275} C_DIS
LIN {X 68.9821,Y 59.5955,Z 93,A 36.517,B 24.9077,C -2.2176,E1 25.1193,E2 408.4376} C_DIS
LIN {X 65.7878,Y 63.1025,Z 93,A 39.1141,B 24.9083,C -2.2104,E1 25.1144,E2 405.8689} C_DIS
LIN {X 63.2245,Y 65.6702,Z 93,A 41.3964,B 24.9079,C -2.2153,E1 25.1098,E2 403.5847} C_DIS
LIN {X 60.5593,Y 68.1366,Z 93,A 43.702,B 24.9075,C -2.2207,E1 25.1051,E2 401.2756} C_DIS
LIN {X 57.9253,Y 70.3901,Z 93,A 46.2375,B 24.9061,C -2.2375,E1 25.0996,E2 398.7101} C_DIS
LIN {X 54.0348,Y 73.418,Z 93,A 48.9165,B 24.9069,C -2.2281,E1 25.0937,E2 396.0629} C_DIS
LIN {X 51.1675,Y 75.4441,Z 93,A 50.9433,B 24.9071,C -2.2255,E1 25.089,E2 394.0493} C_DIS
LIN {X 48.5024,Y 77.1848,Z 93,A 52.8184,B 24.9071,C -2.2243,E1 25.0847,E2 392.1832} C_DIS
LIN {X 45.3024,Y 79.1051,Z 93,A 55.3853,B 24.9063,C -2.2354,E1 25.0785,E2 389.5979} C_DIS
LIN {X 43.3088,Y 80.214,Z 93,A 57.2789,B 24.9047,C -2.2533,E1 25.0737,E2 387.6673} C_DIS
LIN {X 39.3992,Y 82.2048,Z 93,A 59.5008,B 24.906,C -2.2381,E1 25.0682,E2 385.4873} C_DIS
LIN {X 36.0285,Y 83.738,Z 93,A 62.1736,B 24.9048,C -2.2526,E1 25.0613,E2 382.7867} C_DIS
LIN {X 33.2981,Y 84.8596,Z 93,A 64.204,B 24.9041,C -2.2605,E1 25.056,E2 380.7421} C_DIS
LIN {X 28.6654,Y 86.5358,Z 93,A 66.9455,B 24.905,C -2.2509,E1 25.0489,E2 378.0287} C_DIS
LIN {X 25.5883,Y 87.4944,Z 93,A 68.9544,B 24.9049,C -2.2518,E1 25.0435,E2 376.0211} C_DIS
LIN {X 22.0714,Y 88.4477,Z 93,A 71.2216,B 24.9049,C -2.2525,E1 25.0374,E2 373.756} C_DIS
LIN {X 19.0114,Y 89.1552,Z 93,A 73.6365,B 24.9035,C -2.2684,E1 25.0307,E2 371.3065} C_DIS
LIN {X 15.7436,Y 89.7898,Z 93,A 75.1663,B 24.905,C -2.2502,E1 25.0266,E2 369.8215} C_DIS
LIN {X 12.3678,Y 90.317,Z 93,A 77.3694,B 24.9048,C -2.2526,E1 25.0205,E2 367.6147} C_DIS
LIN {X 8.3434,Y 90.7761,Z 93,A 79.8339,B 24.905,C -2.2503,E1 25.0137,E2 365.1574} C_DIS
LIN {X 3.6044,Y 91.088,Z 93,A 82.8664,B 24.9049,C -2.2518,E1 25.0052,E2 362.1224} C_DIS
LIN {X 0.4094,Y 91.1579,Z 93,A 84.6738,B 24.9055,C -2.2449,E1 25.0002,E2 360.3317} C_DIS
LIN {X -1.6379,Y 91.144,Z 93,A 86.3975,B 24.9043,C -2.2589,E1 24.9953,E2 358.5745} C_DIS
LIN {X -6.4341,Y 90.9318,Z 93,A 89.3051,B 24.9047,C -2.2542,E1 24.9872,E2 355.6773} C_DIS
LIN {X -10.1037,Y 90.5985,Z 93,A 91.4161,B 24.9053,C -2.2463,E1 24.9814,E2 353.5839} C_DIS
LIN {X -14.325,Y 90.027,Z 93,A 94.0652,B 24.9056,C -2.2436,E1 24.9741,E2 350.939} C_DIS
LIN {X -17.964,Y 89.372,Z 93,A 96.445,B 24.9056,C -2.2436,E1 24.9676,E2 348.5567} C_DIS
LIN {X -21.0089,Y 88.7062,Z 93,A 98.6468,B 24.9051,C -2.2497,E1 24.9615,E2 346.3376} C_DIS
LIN {X -24.6372,Y 87.7666,Z 93,A 101.2333,B 24.9046,C -2.2547,E1 24.9545,E2 343.7351} C_DIS
LIN {X -29.0657,Y 86.4008,Z 93,A 104.0175,B 24.9053,C -2.2472,E1 24.9472,E2 340.9639} C_DIS
LIN {X -33.141,Y 84.9213,Z 93,A 106.5546,B 24.9061,C -2.2376,E1 24.9406,E2 338.4443} C_DIS
LIN {X -36.41,Y 83.5717,Z 93,A 108.7459,B 24.9064,C -2.2334,E1 24.935,E2 336.2579} C_DIS
LIN {X -39.8082,Y 82.0083,Z 93,A 111.1133,B 24.9067,C -2.2303,E1 24.929,E2 333.8919} C_DIS
LIN {X -42.5245,Y 80.6324,Z 93,A 112.9871,B 24.9071,C -2.2259,E1 24.9244,E2 332.0235} C_DIS
LIN {X -45.9707,Y 78.72,Z 93,A 115.4917,B 24.9074,C -2.2224,E1 24.9183,E2 329.5198} C_DIS
LIN {X -49.1309,Y 76.7855,Z 93,A 118.4227,B 24.9061,C -2.237,E1 24.9112,E2 326.5448} C_DIS
LIN {X -52.0816,Y 74.816,Z 93,A 120.3914,B 24.9072,C -2.2243,E1 24.9068,E2 324.5996} C_DIS
LIN {X -55.0678,Y 72.6472,Z 93,A 122.3032,B 24.9086,C -2.2068,E1 24.9026,E2 322.7227} C_DIS
LIN {X -57.6722,Y 70.5971,Z 93,A 124.6025,B 24.9085,C -2.209,E1 24.8975,E2 320.4095} C_DIS
LIN {X -60.4068,Y 68.2731,Z 93,A 126.874,B 24.9088,C -2.2044,E1 24.8927,E2 318.14} C_DIS
LIN {X -62.9158,Y 65.9677,Z 93,A 128.8321,B 24.9097,C -2.1938,E1 24.8888,E2 316.1993} C_DIS
LIN {X -64.9785,Y 63.9354,Z 93,A 130.862,B 24.9096,C -2.1959,E1 24.8848,E2 314.1559} C_DIS
LIN {X -67.3298,Y 61.4547,Z 93,A 132.9853,B 24.9101,C -2.1898,E1 24.8807,E2 312.0377} C_DIS
LIN {X -69.6767,Y 58.7815,Z 93,A 135.2249,B 24.9105,C -2.1842,E1 24.8767,E2 309.8014} C_DIS
LIN {X -71.822,Y 56.1404,Z 93,A 137.3729,B 24.911,C -2.1788,E1 24.8729,E2 307.6561} C_DIS
LIN {X -73.4201,Y 54.032,Z 93,A 139.7084,B 24.9096,C -2.195,E1 24.869,E2 305.2707} C_DIS
LIN {X -75.7462,Y 50.7213,Z 93,A 142.349,B 24.91,C -2.1909,E1 24.8649,E2 302.6266} C_DIS
LIN {X -78.0244,Y 47.1399,Z 93,A 145.1776,B 24.9102,C -2.1883,E1 24.8608,E2 299.7897} C_DIS
LIN {X -80.4085,Y 42.9497,Z 93,A 147.4724,B 24.9127,C -2.1569,E1 24.8578,E2 297.5576} C_DIS
LIN {X -82.6294,Y 38.5007,Z 93,A 150.3747,B 24.914,C -2.1409,E1 24.8543,E2 294.6778} C_DIS
LIN {X -83.9545,Y 35.5185,Z 93,A 152.4884,B 24.9144,C -2.1366,E1 24.852,E2 292.5626} C_DIS
LIN {X -85.2548,Y 32.2728,Z 93,A 154.7936,B 24.9147,C -2.1332,E1 24.8496,E2 290.2529} C_DIS
LIN {X -86.2035,Y 29.6508,Z 93,A 156.6948,B 24.9147,C -2.1322,E1 24.8479,E2 288.3431} C_DIS
LIN {X -87.7308,Y 24.7634,Z 93,A 159.7225,B 24.916,C -2.1164,E1 24.8454,E2 285.3357} C_DIS
LIN {X -88.5499,Y 21.6524,Z 93,A 161.7175,B 24.9166,C -2.1092,E1 24.8441,E2 283.3462} C_DIS
LIN {X -89.227,Y 18.6702,Z 93,A 163.4307,B 24.9175,C -2.0969,E1 24.8431,E2 281.6524} C_DIS
LIN {X -89.7661,Y 15.8755,Z 93,A 165.7791,B 24.9167,C -2.108,E1 24.8419,E2 279.2636} C_DIS
LIN {X -90.3992,Y 11.7429,Z 93,A 168.1059,B 24.918,C -2.0905,E1 24.841,E2 276.9646} C_DIS
LIN {X -90.7409,Y 8.7248,Z 93,A 170.1528,B 24.9182,C -2.0885,E1 24.8404,E2 274.9102} C_DIS
LIN {X -91.0085,Y 5.2349,Z 93,A 172.299,B 24.9189,C -2.0798,E1 24.84,E2 272.7717} C_DIS
LIN {X -91.1508,Y 1.2703,Z 93,A 174.7256,B 24.9197,C -2.0698,E1 24.8398,E2 270.3545} C_DIS
LIN {X -91.1393,Y -1.8957,Z 93,A 176.8822,B 24.9197,C -2.0685,E1 24.8398,E2 268.1881} C_DIS
LIN {X -90.9133,Y -6.7073,Z 93,A 179.7082,B 24.921,C -2.0527,E1 24.8403,E2 265.3826} C_DIS
LIN {X -90.6352,Y -9.7592,Z 93,A -178.1257,B 24.9209,C -2.0539,E1 24.8409,E2 263.2009} C_DIS
LIN {X -90.1944,Y -13.2309,Z 93,A -175.941,B 24.9215,C -2.0465,E1 24.8417,E2 261.0206} C_DIS
LIN {X -89.6432,Y -16.5588,Z 93,A -173.7839,B 24.9219,C -2.041,E1 24.8428,E2 258.8639} C_DIS
LIN {X -88.937,Y -20.0097,Z 93,A -171.5938,B 24.9225,C -2.0334,E1 24.8441,E2 256.679} C_DIS
LIN {X -88.1997,Y -23.0402,Z 93,A -169.7275,B 24.9231,C -2.0246,E1 24.8453,E2 254.8228} C_DIS
LIN {X -87.2858,Y -26.2914,Z 93,A -167.4647,B 24.9233,C -2.0225,E1 24.8471,E2 252.552} C_DIS
LIN {X -85.8826,Y -30.5633,Z 93,A -164.4203,B 24.9234,C -2.0208,E1 24.8499,E2 249.4944} C_DIS
LIN {X -83.7495,Y -36.002,Z 93,A -161.0937,B 24.925,C -1.9996,E1 24.8533,E2 246.1998} C_DIS
LIN {X -82.6131,Y -38.5356,Z 93,A -159.2976,B 24.9253,C -1.9962,E1 24.8554,E2 244.4018} C_DIS
LIN {X -81.0307,Y -41.7617,Z 93,A -156.9115,B 24.9255,C -1.9939,E1 24.8584,E2 242.0085} C_DIS
LIN {X -79.6984,Y -44.2507,Z 93,A -154.8297,B 24.9251,C -1.9986,E1 24.8612,E2 239.9046} C_DIS
LIN {X -77.4997,Y -47.9983,Z 93,A -152.1146,B 24.9257,C -1.9909,E1 24.8652,E2 237.1938} C_DIS
LIN {X -75.1563,Y -51.5919,Z 93,A -149.5333,B 24.9265,C -1.9805,E1 24.8692,E2 234.6245} C_DIS
LIN {X -73.3967,Y -54.064,Z 93,A -147.4423,B 24.9264,C -1.9815,E1 24.8726,E2 232.5209} C_DIS
LIN {X -70.4447,Y -57.8595,Z 93,A -144.6618,B 24.9275,C -1.9668,E1 24.8774,E2 229.7624} C_DIS
LIN {X -66.2795,Y -62.5857,Z 93,A -140.6844,B 24.9281,C -1.9585,E1 24.8849,E2 225.7871} C_DIS
LIN {X -63.7323,Y -65.1791,Z 93,A -138.4915,B 24.9287,C -1.9508,E1 24.8892,E2 223.6033} C_DIS
LIN {X -61.1537,Y -67.6044,Z 93,A -136.3204,B 24.9291,C -1.9446,E1 24.8936,E2 221.438} C_DIS
LIN {X -59.1283,Y -69.3813,Z 93,A -134.1219,B 24.9282,C -1.9574,E1 24.8984,E2 219.2005} C_DIS
LIN {X -54.1295,Y -73.3486,Z 93,A -130.4551,B 24.9295,C -1.9393,E1 24.9064,E2 215.5637} C_DIS
LIN {X -50.5946,Y -75.831,Z 93,A -127.3616,B 24.9289,C -1.947,E1 24.9136,E2 212.4413} C_DIS
LIN {X -46.6127,Y -78.3406,Z 93,A -124.4483,B 24.9294,C -1.9412,E1 24.9206,E2 209.5328} C_DIS
LIN {X -42.8244,Y -80.4744,Z 93,A -121.9873,B 24.9303,C -1.9287,E1 24.9265,E2 207.0945} C_DIS
LIN {X -39.8038,Y -82.0104,Z 93,A -120.0392,B 24.9309,C -1.9202,E1 24.9314,E2 205.1614} C_DIS
LIN {X -36.5745,Y -83.5,Z 93,A -117.1876,B 24.9296,C -1.9379,E1 24.9388,E2 202.2609} C_DIS
LIN {X -33.4721,Y -84.7913,Z 93,A -115.7318,B 24.9313,C -1.9143,E1 24.9424,E2 200.858} C_DIS
LIN {X -30.1357,Y -86.0335,Z 93,A -113.401,B 24.9313,C -1.9154,E1 24.9485,E2 198.52} C_DIS
LIN {X -27.3273,Y -86.9669,Z 93,A -111.4699,B 24.9312,C -1.9163,E1 24.9537,E2 196.5832} C_DIS
LIN {X -24.3458,Y -87.8491,Z 93,A -109.4953,B 24.9312,C -1.9157,E1 24.959,E2 194.6069} C_DIS
LIN {X -20.7621,Y -88.7632,Z 93,A -107.1282,B 24.9312,C -1.9158,E1 24.9654,E2 192.2361} C_DIS
LIN {X -16.9763,Y -89.5644,Z 93,A -104.7381,B 24.9314,C -1.9134,E1 24.972,E2 189.849} C_DIS
LIN {X -13.8291,Y -90.1037,Z 93,A -102.5052,B 24.9309,C -1.9205,E1 24.9782,E2 187.5974} C_DIS
LIN {X -10.0115,Y -90.6085,Z 93,A -99.5779,B 24.9296,C -1.9373,E1 24.9864,E2 184.6282} C_DIS
LIN {X -5.8783,Y -90.9694,Z 93,A -97.7697,B 24.9316,C -1.9101,E1 24.9913,E2 182.8838} C_DIS
LIN {X -0.908,Y -91.1549,Z 93,A -94.6575,B 24.9316,C -1.9101,E1 25,E2 179.7714} C_DIS
LIN {X -0.908,Y -91.1549,Z 93,A -94.6575,B 24.9316,C -1.9101,E1 25,E2 179.7714} C_DIS
Enddeposition()
LIN {X 0.5904,Y -90.202,Z 93,A -94.2276,B 24.9316,C -1.9096,E1 25.0012,E2 179.3425} C_DIS
Startdeposition()
$VEL.CP = VEL_PRINT
LIN {X -2.5804,Y -90.1772,Z 93,A -96.6653,B 24.9327,C -1.8951,E1 24.9942,E2 181.8149} C_DIS
LIN {X -5.6931,Y -90.0349,Z 93,A -98.4991,B 24.9323,C -1.8997,E1 24.9892,E2 183.6382} C_DIS
LIN {X -8.8486,Y -89.78,Z 93,A -100.6538,B 24.9327,C -1.8951,E1 24.9831,E2 185.8049} C_DIS
LIN {X -11.326,Y -89.5005,Z 93,A -102.2663,B 24.9327,C -1.8944,E1 24.9787,E2 187.4202} C_DIS
LIN {X -15.0755,Y -88.9456,Z 93,A -104.6648,B 24.9327,C -1.8954,E1 24.972,E2 189.8186} C_DIS
LIN {X -18.5452,Y -88.2881,Z 93,A -106.9077,B 24.9326,C -1.8962,E1 24.9659,E2 192.0619} C_DIS
LIN {X -21.7566,Y -87.5519,Z 93,A -108.8129,B 24.9321,C -1.9034,E1 24.9608,E2 193.9527} C_DIS
LIN {X -24.4515,Y -86.8371,Z 93,A -110.7331,B 24.9323,C -1.8997,E1 24.9555,E2 195.8847} C_DIS
LIN {X -27.3009,Y -85.9852,Z 93,A -112.6969,B 24.9324,C -1.8986,E1 24.9503,E2 197.8544} C_DIS
LIN {X -30.5236,Y -84.8942,Z 93,A -114.8869,B 24.9324,C -1.8995,E1 24.9445,E2 200.0465} C_DIS
LIN {X -34.5489,Y -83.3378,Z 93,A -117.549,B 24.932,C -1.9047,E1 24.9376,E2 202.7021} C_DIS
LIN {X -37.4522,Y -82.0735,Z 93,A -119.6708,B 24.932,C -1.9034,E1 24.9322,E2 204.8321} C_DIS
LIN {X -40.7708,Y -80.476,Z 93,A -121.9154,B 24.9317,C -1.9092,E1 24.9266,E2 207.0687} C_DIS
LIN {X -43.7558,Y -78.8926,Z 93,A -123.7762,B 24.9308,C -1.921,E1 24.9221,E2 208.9067} C_DIS
LIN {X -46.3355,Y -77.4068,Z 93,A -125.9224,B 24.9312,C -1.9157,E1 24.9169,E2 211.072} C_DIS
LIN {X -49.2985,Y -75.5539,Z 93,A -128.2231,B 24.9312,C -1.9166,E1 24.9114,E2 213.378} C_DIS
LIN {X -51.6749,Y -73.948,Z 93,A -130.0215,B 24.9309,C -1.9203,E1 24.9073,E2 215.1738} C_DIS
LIN {X -53.6667,Y -72.5165,Z 93,A -132.1653,B 24.932,C -1.9049,E1 24.9024,E2 217.3616} C_DIS
LIN {X -56.517,Y -70.3172,Z 93,A -134.5804,B 24.932,C -1.9052,E1 24.8971,E2 219.7851} C_DIS
LIN {X -59.5918,Y -67.7308,Z 93,A -136.6396,B 24.9305,C -1.9251,E1 24.8929,E2 221.805} C_DIS
LIN {X -62.6469,Y -64.9146,Z 93,A -139.005,B 24.9295,C -1.9389,E1 24.8881,E2 224.1474} C_DIS
LIN {X -64.9619,Y -62.5979,Z 93,A -140.9865,B 24.929,C -1.9463,E1 24.8842,E2 226.1197} C_DIS
LIN {X -67.8844,Y -59.416,Z 93,A -144.4558,B 24.9301,C -1.9305,E1 24.8777,E2 229.642} C_DIS
LIN {X -70.07,Y -56.822,Z 93,A -145.6305,B 24.9276,C -1.9651,E1 24.8757,E2 230.7398} C_DIS
LIN {X -72.3449,Y -53.897,Z 93,A -148.5031,B 24.9283,C -1.955,E1 24.8708,E2 233.6501} C_DIS
LIN {X -74.329,Y -51.1267,Z 93,A -150.632,B 24.9279,C -1.9614,E1 24.8673,E2 235.774} C_DIS
LIN {X -76.175,Y -48.3336,Z 93,A -152.7383,B 24.9274,C -1.9675,E1 24.8641,E2 237.8765} C_DIS
LIN {X -77.6544,Y -45.9167,Z 93,A -154.5047,B 24.927,C -1.9732,E1 24.8616,E2 239.6383} C_DIS
LIN {X -79.0856,Y -43.4074,Z 93,A -156.4755,B 24.927,C -1.9741,E1 24.8589,E2 241.6174} C_DIS
LIN {X -80.4886,Y -40.7462,Z 93,A -158.4319,B 24.9266,C -1.978,E1 24.8564,E2 243.575} C_DIS
LIN {X -82.0695,Y -37.4609,Z 93,A -160.5162,B 24.9256,C -1.9913,E1 24.8539,E2 245.6387} C_DIS
LIN {X -83.1708,Y -34.9452,Z 93,A -162.3386,B 24.9254,C -1.994,E1 24.8519,E2 247.4649} C_DIS
LIN {X -84.2224,Y -32.3311,Z 93,A -165.0231,B 24.927,C -1.973,E1 24.8492,E2 250.2146} C_DIS
LIN {X -85.6513,Y -28.3293,Z 93,A -167.0455,B 24.9249,C -2.0007,E1 24.8474,E2 252.1824} C_DIS
LIN {X -86.3996,Y -25.9566,Z 93,A -168.5409,B 24.9244,C -2.0079,E1 24.8462,E2 253.6691} C_DIS
LIN {X -87.2785,Y -22.8286,Z 93,A -170.6397,B 24.924,C -2.0131,E1 24.8447,E2 255.7678} C_DIS
LIN {X -88.0873,Y -19.4742,Z 93,A -172.897,B 24.9236,C -2.018,E1 24.8432,E2 258.0268} C_DIS
LIN {X -88.7989,Y -15.9157,Z 93,A -175.1332,B 24.9229,C -2.0271,E1 24.8421,E2 260.2544} C_DIS
LIN {X -89.3398,Y -12.5288,Z 93,A -177.2424,B 24.9223,C -2.036,E1 24.8412,E2 262.355} C_DIS
LIN {X -89.7478,Y -9.1616,Z 93,A -179.4717,B 24.9219,C -2.0406,E1 24.8405,E2 264.5867} C_DIS
LIN {X -90.0158,Y -5.9752,Z 93,A 178.5026,B 24.9214,C -2.0472,E1 24.8401,E2 266.6088} C_DIS
LIN {X -90.169,Y -2.8469,Z 93,A 176.4534,B 24.9211,C -2.0518,E1 24.8398,E2 268.6593} C_DIS
LIN {X -90.2125,Y 0.5969,Z 93,A 174.2242,B 24.9206,C -2.0575,E1 24.8398,E2 270.8882} C_DIS
LIN {X -90.1507,Y 3.4065,Z 93,A 172.3609,B 24.9203,C -2.061,E1 24.84,E2 272.7545} C_DIS
LIN {X -89.9434,Y 6.9831,Z 93,A 170.3918,B 24.9191,C -2.0772,E1 24.8403,E2 274.6967} C_DIS
LIN {X -89.7687,Y 8.962,Z 93,A 168.7945,B 24.9195,C -2.0715,E1 24.8407,E2 276.3173} C_DIS
LIN {X -89.356,Y 12.4144,Z 93,A 166.8241,B 24.9184,C -2.0855,E1 24.8414,E2 278.266} C_DIS
LIN {X -88.9737,Y 14.9073,Z 93,A 165.1153,B 24.9183,C -2.0875,E1 24.8422,E2 279.9802} C_DIS
LIN {X -88.3903,Y 18.047,Z 93,A 163.1524,B 24.9176,C -2.0958,E1 24.8432,E2 281.9348} C_DIS
LIN {X -87.7922,Y 20.7677,Z 93,A 161.3641,B 24.9172,C -2.1009,E1 24.8443,E2 283.7216} C_DIS
LIN {X -87.109,Y 23.4642,Z 93,A 159.6933,B 24.9166,C -2.1092,E1 24.8455,E2 285.3821} C_DIS
LIN {X -85.4481,Y 28.934,Z 93,A 155.8945,B 24.9161,C -2.1156,E1 24.8486,E2 289.1876} C_DIS
LIN {X -84.1563,Y 32.5041,Z 93,A 153.4568,B 24.9155,C -2.1222,E1 24.851,E2 291.6233} C_DIS
LIN {X -83.1025,Y 35.1074,Z 93,A 151.5183,B 24.9155,C -2.1231,E1 24.8531,E2 293.5704} C_DIS
LIN {X -81.7057,Y 38.246,Z 93,A 149.3705,B 24.9149,C -2.1307,E1 24.8555,E2 295.712} C_DIS
LIN {X -79.4403,Y 42.7537,Z 93,A 146.0878,B 24.9143,C -2.1378,E1 24.8597,E2 298.9953} C_DIS
LIN {X -77.7911,Y 45.6854,Z 93,A 143.986,B 24.9137,C -2.1449,E1 24.8626,E2 301.0909} C_DIS
LIN {X -75.986,Y 48.628,Z 93,A 141.8562,B 24.9131,C -2.153,E1 24.8658,E2 303.2124} C_DIS
LIN {X -72.562,Y 53.6046,Z 93,A 137.8292,B 24.9127,C -2.1578,E1 24.8723,E2 307.2476} C_DIS
LIN {X -70.4156,Y 56.3955,Z 93,A 135.5776,B 24.9122,C -2.1633,E1 24.8761,E2 309.4969} C_DIS
LIN {X -68.0659,Y 59.2082,Z 93,A 133.3055,B 24.9116,C -2.1709,E1 24.8802,E2 311.7612} C_DIS
LIN {X -65.8094,Y 61.7064,Z 93,A 131.1782,B 24.9111,C -2.1765,E1 24.8842,E2 313.8843} C_DIS
LIN {X -63.5856,Y 63.9959,Z 93,A 129.1343,B 24.9108,C -2.1809,E1 24.8882,E2 315.9265} C_DIS
LIN {X -61.0895,Y 66.3824,Z 93,A 126.9394,B 24.9104,C -2.186,E1 24.8927,E2 318.1183} C_DIS
LIN {X -58.6358,Y 68.5596,Z 93,A 124.8977,B 24.9099,C -2.192,E1 24.897,E2 320.1539} C_DIS
LIN {X -56.0952,Y 70.6534,Z 93,A 122.7821,B 24.9096,C -2.1958,E1 24.9016,E2 322.2684} C_DIS
LIN {X -53.9453,Y 72.3086,Z 93,A 120.8262,B 24.9098,C -2.1923,E1 24.906,E2 324.2394} C_DIS
LIN {X -50.7092,Y 74.6133,Z 93,A 118.35,B 24.9093,C -2.1988,E1 24.9116,E2 326.7087} C_DIS
LIN {X -46.6704,Y 77.204,Z 93,A 115.546,B 24.9082,C -2.2119,E1 24.9182,E2 329.4904} C_DIS
LIN {X -43.2494,Y 79.1714,Z 93,A 112.8716,B 24.9082,C -2.2111,E1 24.9247,E2 332.1744} C_DIS
LIN {X -40.4027,Y 80.6617,Z 93,A 110.8092,B 24.9081,C -2.2138,E1 24.9298,E2 334.2361} C_DIS
LIN {X -37.2161,Y 82.1799,Z 93,A 108.5969,B 24.9077,C -2.2181,E1 24.9354,E2 336.4436} C_DIS
LIN {X -34.2252,Y 83.4699,Z 93,A 106.5139,B 24.9075,C -2.2206,E1 24.9408,E2 338.5254} C_DIS
LIN {X -31.0063,Y 84.7181,Z 93,A 104.5279,B 24.9067,C -2.2299,E1 24.9459,E2 340.4935} C_DIS
LIN {X -28.2235,Y 85.6867,Z 93,A 102.6429,B 24.9066,C -2.2317,E1 24.9509,E2 342.3777} C_DIS
LIN {X -25.6958,Y 86.477,Z 93,A 100.8873,B 24.9066,C -2.2314,E1 24.9556,E2 344.1373} C_DIS
LIN {X -23.0439,Y 87.2225,Z 93,A 98.9238,B 24.907,C -2.2265,E1 24.9609,E2 346.1154} C_DIS
LIN {X -19.6253,Y 88.0543,Z 93,A 96.7034,B 24.9068,C -2.229,E1 24.967,E2 348.3329} C_DIS
LIN {X -17.1785,Y 88.5633,Z 93,A 95.2053,B 24.9065,C -2.2331,E1 24.971,E2 349.8228} C_DIS
LIN {X -14.2226,Y 89.0868,Z 93,A 93.201,B 24.9066,C -2.2313,E1 24.9766,E2 351.8332} C_DIS
LIN {X -10.9941,Y 89.5429,Z 93,A 91.1279,B 24.9066,C -2.2325,E1 24.9823,E2 353.905} C_DIS
LIN {X -7.611,Y 89.8932,Z 93,A 89.012,B 24.9063,C -2.235,E1 24.9882,E2 356.0161} C_DIS
LIN {X -4.7874,Y 90.087,Z 93,A 87.0785,B 24.9066,C -2.2314,E1 24.9936,E2 357.9588} C_DIS
LIN {X -1.3923,Y 90.2035,Z 93,A 84.9829,B 24.9064,C -2.2339,E1 24.9994,E2 360.0485} C_DIS
LIN {X 2.3533,Y 90.1841,Z 93,A 82.6029,B 24.9064,C -2.2342,E1 25.0061,E2 362.4275} C_DIS
LIN {X 6.4192,Y 89.9858,Z 93,A 80.0665,B 24.9062,C -2.2358,E1 25.0131,E2 364.9592} C_DIS
LIN {X 10.0383,Y 89.6548,Z 93,A 77.7229,B 24.9063,C -2.2344,E1 25.0197,E2 367.3047} C_DIS
LIN {X 13.4332,Y 89.2088,Z 93,A 75.7987,B 24.9057,C -2.242,E1 25.0249,E2 369.2092} C_DIS
LIN {X 16.2572,Y 88.7374,Z 93,A 73.8357,B 24.9062,C -2.2366,E1 25.0304,E2 371.1828} C_DIS
LIN {X 19.7165,Y 88.0344,Z 93,A 71.4803,B 24.9066,C -2.2318,E1 25.0368,E2 373.5465} C_DIS
LIN {X 23.2656,Y 87.1626,Z 93,A 69.2288,B 24.9065,C -2.2327,E1 25.0429,E2 375.7925} C_DIS
LIN {X 26.1003,Y 86.357,Z 93,A 67.4454,B 24.9064,C -2.2343,E1 25.0476,E2 377.5691} C_DIS
LIN {X 29.0259,Y 85.4171,Z 93,A 65.7056,B 24.9059,C -2.2398,E1 25.0522,E2 379.2926} C_DIS
LIN {X 31.7677,Y 84.4357,Z 93,A 63.6481,B 24.9066,C -2.2312,E1 25.0577,E2 381.3663} C_DIS
LIN {X 34.6916,Y 83.2777,Z 93,A 61.5866,B 24.907,C -2.227,E1 25.063,E2 383.4331} C_DIS
LIN {X 37.7069,Y 81.9567,Z 93,A 59.4559,B 24.9073,C -2.2233,E1 25.0684,E2 385.5672} C_DIS
LIN {X 40.9569,Y 80.3809,Z 93,A 57.2661,B 24.9073,C -2.2239,E1 25.0739,E2 387.7496} C_DIS
LIN {X 43.9416,Y 78.7888,Z 93,A 55.2912,B 24.907,C -2.2269,E1 25.0787,E2 389.7118} C_DIS
LIN {X 47.0692,Y 76.9617,Z 93,A 52.926,B 24.9074,C -2.2213,E1 25.0844,E2 392.0829} C_DIS
LIN {X 49.0761,Y 75.6984,Z 93,A 51.2567,B 24.9081,C -2.2134,E1 25.0884,E2 393.7655} C_DIS
LIN {X 51.3074,Y 74.2034,Z 93,A 49.5867,B 24.9082,C -2.2118,E1 25.0922,E2 395.4336} C_DIS
LIN {X 54.1545,Y 72.1515,Z 93,A 47.3574,B 24.9086,C -2.2079,E1 25.0972,E2 397.6642} C_DIS
LIN {X 57.2423,Y 69.7291,Z 93,A 44.8918,B 24.9089,C -2.2043,E1 25.1026,E2 400.1292} C_DIS
LIN {X 59.6514,Y 67.6788,Z 93,A 42.7974,B 24.9094,C -2.1974,E1 25.1071,E2 402.2316} C_DIS
LIN {X 62.1186,Y 65.4218,Z 93,A 40.6742,B 24.9098,C -2.1931,E1 25.1114,E2 404.3563} C_DIS
LIN {X 64.7257,Y 62.8429,Z 93,A 38.4996,B 24.9098,C -2.1935,E1 25.1157,E2 406.5208} C_DIS
LIN {X 66.8455,Y 60.5848,Z 93,A 36.3304,B 24.9107,C -2.1821,E1 25.1198,E2 408.7073} C_DIS
LIN {X 69.3944,Y 57.6451,Z 93,A 33.9842,B 24.9107,C -2.1807,E1 25.124,E2 411.046} C_DIS
LIN {X 71.6208,Y 54.855,Z 93,A 31.7095,B 24.9113,C -2.175,E1 25.1279,E2 413.3235} C_DIS
LIN {X 73.6452,Y 52.1062,Z 93,A 29.0351,B 24.9131,C -2.152,E1 25.1323,E2 416.0394} C_DIS
LIN {X 75.6833,Y 49.0996,Z 93,A 27.16,B 24.9124,C -2.1611,E1 25.1352,E2 417.8836} C_DIS
LIN {X 77.7538,Y 45.7485,Z 93,A 24.9687,B 24.912,C -2.1655,E1 25.1383,E2 420.0534} C_DIS
LIN {X 79.3891,Y 42.8479,Z 93,A 22.7982,B 24.9127,C -2.1578,E1 25.1413,E2 422.2307} C_DIS
LIN {X 80.8211,Y 40.0811,Z 93,A 20.776,B 24.9132,C -2.1508,E1 25.1438,E2 424.2587} C_DIS
LIN {X 81.8567,Y 37.9216,Z 93,A 18.7395,B 24.915,C -2.1283,E1 25.1463,E2 426.3373} C_DIS
LIN {X 83.2204,Y 34.8269,Z 93,A 17.264,B 24.9136,C -2.1459,E1 25.1478,E2 427.7631} C_DIS
LIN {X 84.2291,Y 32.3133,Z 93,A 15.3994,B 24.9144,C -2.1357,E1 25.1497,E2 429.6414} C_DIS
LIN {X 85.3885,Y 29.1107,Z 93,A 13.2307,B 24.915,C -2.1292,E1 25.1517,E2 431.8134} C_DIS
LIN {X 86.4626,Y 25.7443,Z 93,A 11.0236,B 24.9154,C -2.1238,E1 25.1536,E2 434.0207} C_DIS
LIN {X 87.4199,Y 22.2785,Z 93,A 8.686,B 24.9161,C -2.1149,E1 25.1552,E2 436.3658} C_DIS
LIN {X 88.3118,Y 18.4296,Z 93,A 6.4345,B 24.916,C -2.1164,E1 25.1566,E2 438.6008} C_DIS
LIN {X 88.8686,Y 15.528,Z 93,A 4.4559,B 24.9168,C -2.1068,E1 25.1576,E2 440.5902} C_DIS
LIN {X 89.4161,Y 11.9776,Z 93,A 1.9932,B 24.9178,C -2.0932,E1 25.1586,E2 443.0707} C_DIS
LIN {X 89.8496,Y 8.1015,Z 93,A -1.0248,B 24.92,C -2.066,E1 25.1594,E2 446.1348} C_DIS
LIN {X 90.1223,Y 4.0688,Z 93,A -2.8197,B 24.9184,C -2.0854,E1 25.1597,E2 447.8733} C_DIS
LIN {X 90.1992,Y 1.6289,Z 93,A -4.7315,B 24.9198,C -2.0675,E1 25.1597,E2 449.816} C_DIS
LIN {X 90.1485,Y -3.4599,Z 93,A -7.6372,B 24.9198,C -2.0688,E1 25.1597,E2 452.7014} C_DIS
LIN {X 89.978,Y -6.5348,Z 93,A -9.4471,B 24.9198,C -2.0678,E1 25.1593,E2 454.5029} C_DIS
LIN {X 89.6848,Y -9.7631,Z 93,A -11.8649,B 24.9213,C -2.0483,E1 25.1586,E2 456.9525} C_DIS
LIN {X 89.0666,Y -14.3514,Z 93,A -14.3591,B 24.9208,C -2.0549,E1 25.1576,E2 459.4164} C_DIS
LIN {X 88.6141,Y -16.9148,Z 93,A -16.118,B 24.9215,C -2.0458,E1 25.1567,E2 461.1865} C_DIS
LIN {X 87.9706,Y -19.9954,Z 93,A -18.1369,B 24.9221,C -2.0387,E1 25.1555,E2 463.2103} C_DIS
LIN {X 87.2848,Y -22.8042,Z 93,A -19.764,B 24.9219,C -2.0404,E1 25.1544,E2 464.824} C_DIS
LIN {X 86.4387,Y -25.8249,Z 93,A -22.038,B 24.9232,C -2.024,E1 25.1527,E2 467.1236} C_DIS
LIN {X 85.3306,Y -29.2823,Z 93,A -24.0694,B 24.923,C -2.0267,E1 25.1509,E2 469.1373} C_DIS
LIN {X 84.5226,Y -31.5367,Z 93,A -26.0705,B 24.9246,C -2.0048,E1 25.1489,E2 471.1789} C_DIS
LIN {X 82.8929,Y -35.6026,Z 93,A -28.5761,B 24.9246,C -2.0062,E1 25.1462,E2 473.6674} C_DIS
LIN {X 81.6442,Y -38.3781,Z 93,A -30.5109,B 24.925,C -2.0003,E1 25.144,E2 475.6056} C_DIS
LIN {X 80.3501,Y -41.0171,Z 93,A -32.7562,B 24.9264,C -1.9813,E1 25.1411,E2 477.8838} C_DIS
LIN {X 78.8358,Y -43.8575,Z 93,A -34.315,B 24.9256,C -1.9926,E1 25.1391,E2 479.4077} C_DIS
LIN {X 77.1189,Y -46.8105,Z 93,A -36.2635,B 24.9254,C -1.9943,E1 25.1363,E2 481.3422} C_DIS
LIN {X 75.5757,Y -49.2654,Z 93,A -38.381,B 24.9266,C -1.9792,E1 25.1331,E2 483.4848} C_DIS
LIN {X 73.5768,Y -52.202,Z 93,A -40.5778,B 24.9269,C -1.9751,E1 25.1296,E2 485.6804} C_DIS
LIN {X 71.4917,Y -55.0226,Z 93,A -42.5985,B 24.9268,C -1.9765,E1 25.1262,E2 487.6882} C_DIS
LIN {X 69.5825,Y -57.4187,Z 93,A -44.7668,B 24.9277,C -1.9634,E1 25.1224,E2 489.8773} C_DIS
LIN {X 67.1935,Y -60.1962,Z 93,A -46.9799,B 24.9279,C -1.9615,E1 25.1183,E2 492.085} C_DIS
LIN {X 64.9049,Y -62.657,Z 93,A -49.0911,B 24.9282,C -1.957,E1 25.1143,E2 494.1977} C_DIS
LIN {X 62.4717,Y -65.0836,Z 93,A -51.2739,B 24.9286,C -1.9517,E1 25.1099,E2 496.3838} C_DIS
LIN {X 59.9872,Y -67.3805,Z 93,A -53.4208,B 24.9289,C -1.9468,E1 25.1055,E2 498.5337} C_DIS
LIN {X 57.521,Y -69.4976,Z 93,A -55.3462,B 24.9289,C -1.947,E1 25.1014,E2 500.451} C_DIS
LIN {X 55.6863,Y -70.9766,Z 93,A -56.9774,B 24.9295,C -1.9391,E1 25.0978,E2 502.095} C_DIS
LIN {X 53.0875,Y -72.9406,Z 93,A -59.1005,B 24.93,C -1.9328,E1 25.093,E2 504.2252} C_DIS
LIN {X 50.7738,Y -74.5696,Z 93,A -60.8356,B 24.93,C -1.9314,E1 25.089,E2 505.9579} C_DIS
LIN {X 47.9171,Y -76.4363,Z 93,A -62.8189,B 24.93,C -1.9336,E1 25.0844,E2 507.9294} C_DIS
LIN {X 45.798,Y -77.7245,Z 93,A -64.6014,B 24.9306,C -1.9235,E1 25.0801,E2 509.7302} C_DIS
LIN {X 42.9052,Y -79.3581,Z 93,A -67.4724,B 24.9328,C -1.8937,E1 25.0729,E2 512.6636} C_DIS
LIN {X 39.0201,Y -81.3387,Z 93,A -69.4606,B 24.9312,C -1.916,E1 25.068,E2 514.5938} C_DIS
LIN {X 35.6673,Y -82.8647,Z 93,A -71.8295,B 24.9315,C -1.9114,E1 25.062,E2 516.9676} C_DIS
LIN {X 32.2374,Y -84.2579,Z 93,A -74.478,B 24.9325,C -1.898,E1 25.055,E2 519.642} C_DIS
LIN {X 27.8833,Y -85.7967,Z 93,A -77.0155,B 24.9318,C -1.9078,E1 25.0484,E2 522.1514} C_DIS
LIN {X 25.1268,Y -86.6458,Z 93,A -79.2669,B 24.9329,C -1.8915,E1 25.0423,E2 524.4375} C_DIS
LIN {X 21.0326,Y -87.7286,Z 93,A -81.6001,B 24.9323,C -1.9008,E1 25.036,E2 526.7451} C_DIS
LIN {X 17.5741,Y -88.4871,Z 93,A -83.6981,B 24.932,C -1.9039,E1 25.0303,E2 528.8331} C_DIS
LIN {X 15.0831,Y -88.9443,Z 93,A -85.5438,B 24.9327,C -1.8947,E1 25.0252,E2 530.6987} C_DIS
LIN {X 10.9821,Y -89.5443,Z 93,A -88.2027,B 24.9329,C -1.8921,E1 25.0178,E2 533.3616} C_DIS
LIN {X 6.9318,Y -89.9475,Z 93,A -90.6942,B 24.9328,C -1.8939,E1 25.0109,E2 535.8474} C_DIS
LIN {X 3.6293,Y -90.1412,Z 93,A -92.7603,B 24.9328,C -1.8942,E1 25.0051,E2 537.912} C_DIS
LIN {X 0.5904,Y -90.202,Z 93,A -94.2266,B 24.9317,C -1.9092,E1 25.0012,E2 539.3425} C_DIS
Enddeposition()
LIN {X 0.5904,Y -90.202,Z 93,A -94.2266,B 24.9317,C -1.9092,E1 25.0012,E2 539.3425} C_DIS
Startdeposition()
$VEL.CP = VEL_PRINT
LIN {X 1.9606,Y -89.2481,Z 93,A -92.7835,B 24.9291,C -1.9445,E1 25.0054,E2 537.816} C_DIS
LIN {X 5.278,Y -89.1135,Z 93,A -90.8331,B 24.9295,C -1.9393,E1 25.0108,E2 535.8785} C_DIS
LIN {X 7.6487,Y -88.9424,Z 93,A -89.3277,B 24.9295,C -1.9393,E1 25.015,E2 534.3739} C_DIS
LIN {X 9.8218,Y -88.7286,Z 93,A -87.7158,B 24.9289,C -1.9472,E1 25.0195,E2 532.7444} C_DIS
LIN {X 13.0898,Y -88.3057,Z 93,A -85.594,B 24.9288,C -1.9488,E1 25.0254,E2 530.6205} C_DIS
LIN {X 16.1501,Y -87.7967,Z 93,A -83.8097,B 24.9292,C -1.9434,E1 25.0303,E2 528.851} C_DIS
LIN {X 18.2937,Y -87.3752,Z 93,A -82.4096,B 24.9292,C -1.9446,E1 25.0341,E2 527.4499} C_DIS
LIN {X 20.5964,Y -86.862,Z 93,A -80.9176,B 24.9291,C -1.9452,E1 25.0382,E2 525.9584} C_DIS
LIN {X 22.7323,Y -86.3277,Z 93,A -79.5061,B 24.929,C -1.9466,E1 25.042,E2 524.5457} C_DIS
LIN {X 25.4726,Y -85.5577,Z 93,A -77.6031,B 24.9286,C -1.9513,E1 25.0471,E2 522.6349} C_DIS
LIN {X 27.9984,Y -84.7664,Z 93,A -75.9897,B 24.9286,C -1.9504,E1 25.0514,E2 521.0267} C_DIS
LIN {X 29.8848,Y -84.1188,Z 93,A -74.7102,B 24.9286,C -1.952,E1 25.0548,E2 519.7459} C_DIS
LIN {X 31.9571,Y -83.3537,Z 93,A -73.2809,B 24.9284,C -1.9543,E1 25.0585,E2 518.3142} C_DIS
LIN {X 34.5537,Y -82.3105,Z 93,A -71.3893,B 24.928,C -1.9602,E1 25.0634,E2 516.413} C_DIS
LIN {X 36.986,Y -81.2472,Z 93,A -69.7029,B 24.9278,C -1.9622,E1 25.0677,E2 514.7261} C_DIS
LIN {X 39.8333,Y -79.8894,Z 93,A -67.7494,B 24.9278,C -1.963,E1 25.0726,E2 512.7759} C_DIS
LIN {X 42.0409,Y -78.7513,Z 93,A -66.2107,B 24.9278,C -1.9637,E1 25.0764,E2 511.2397} C_DIS
LIN {X 43.9967,Y -77.6759,Z 93,A -64.7776,B 24.9275,C -1.9663,E1 25.0799,E2 509.8048} C_DIS
LIN {X 45.7361,Y -76.6635,Z 93,A -63.4713,B 24.9273,C -1.9691,E1 25.083,E2 508.4957} C_DIS
LIN {X 47.7636,Y -75.4181,Z 93,A -61.9712,B 24.9272,C -1.9711,E1 25.0866,E2 506.9958} C_DIS
LIN {X 49.4354,Y -74.3319,Z 93,A -60.696,B 24.927,C -1.9734,E1 25.0896,E2 505.7192} C_DIS
LIN {X 51.3997,Y -72.9885,Z 93,A -59.1753,B 24.9268,C -1.9763,E1 25.0931,E2 504.1971} C_DIS
LIN {X 53.172,Y -71.7077,Z 93,A -57.5638,B 24.926,C -1.9865,E1 25.0967,E2 502.5671} C_DIS
LIN {X 55.7873,Y -69.6924,Z 93,A -55.4822,B 24.9258,C -1.9898,E1 25.1013,E2 500.4855} C_DIS
LIN {X 58.235,Y -67.6598,Z 93,A -53.4125,B 24.9253,C -1.9953,E1 25.1057,E2 498.4106} C_DIS
LIN {X 60.6799,Y -65.4759,Z 93,A -51.3487,B 24.9251,C -1.9988,E1 25.11,E2 496.3469} C_DIS
LIN {X 63.1107,Y -63.137,Z 93,A -49.198,B 24.9247,C -2.0035,E1 25.1143,E2 494.1942} C_DIS
LIN {X 65.3387,Y -60.8278,Z 93,A -47.1166,B 24.9243,C -2.0094,E1 25.1183,E2 492.1079} C_DIS
LIN {X 67.5281,Y -58.3876,Z 93,A -45.0539,B 24.924,C -2.0133,E1 25.1221,E2 490.0452} C_DIS
LIN {X 69.6864,Y -55.7947,Z 93,A -42.8774,B 24.9235,C -2.0194,E1 25.1259,E2 487.8644} C_DIS
LIN {X 71.7035,Y -53.1776,Z 93,A -40.988,B 24.9237,C -2.0169,E1 25.1291,E2 485.99} C_DIS
LIN {X 72.8724,Y -51.5625,Z 93,A -39.7155,B 24.9235,C -2.0201,E1 25.1311,E2 484.716} C_DIS
LIN {X 74.2217,Y -49.6023,Z 93,A -38.1971,B 24.9232,C -2.024,E1 25.1335,E2 483.1959} C_DIS
LIN {X 75.4143,Y -47.7696,Z 93,A -36.6035,B 24.9224,C -2.0348,E1 25.136,E2 481.5849} C_DIS
LIN {X 77.1279,Y -44.9504,Z 93,A -34.6985,B 24.9224,C -2.0333,E1 25.1387,E2 479.6933} C_DIS
LIN {X 78.112,Y -43.2156,Z 93,A -33.395,B 24.9221,C -2.0379,E1 25.1404,E2 478.3858} C_DIS
LIN {X 79.1592,Y -41.2664,Z 93,A -32.0156,B 24.9219,C -2.0406,E1 25.1422,E2 477.0072} C_DIS
LIN {X 80.1434,Y -39.3208,Z 93,A -30.6251,B 24.9216,C -2.0444,E1 25.144,E2 475.6151} C_DIS
LIN {X 81.1614,Y -37.1764,Z 93,A -29.1112,B 24.9213,C -2.0486,E1 25.1458,E2 474.0994} C_DIS
LIN {X 82.0454,Y -35.1824,Z 93,A -27.7204,B 24.921,C -2.0525,E1 25.1473,E2 472.7069} C_DIS
LIN {X 83.2084,Y -32.3331,Z 93,A -25.7395,B 24.9205,C -2.0588,E1 25.1494,E2 470.7223} C_DIS
LIN {X 84.0381,Y -30.1133,Z 93,A -24.2464,B 24.9202,C -2.0625,E1 25.1508,E2 469.2288} C_DIS
LIN {X 84.7643,Y -28.0047,Z 93,A -22.8263,B 24.9199,C -2.0665,E1 25.1521,E2 467.8072} C_DIS
LIN {X 85.3679,Y -26.1037,Z 93,A -21.537,B 24.9196,C -2.0709,E1 25.1531,E2 466.515} C_DIS
LIN {X 86.0404,Y -23.7971,Z 93,A -20.0306,B 24.9193,C -2.0744,E1 25.1543,E2 465.0088} C_DIS
LIN {X 86.6992,Y -21.2654,Z 93,A -18.2399,B 24.9186,C -2.0838,E1 25.1555,E2 463.2063} C_DIS
LIN {X 87.293,Y -18.6817,Z 93,A -16.6485,B 24.9185,C -2.0852,E1 25.1565,E2 461.6208} C_DIS
LIN {X 87.7239,Y -16.5407,Z 93,A -15.2562,B 24.9181,C -2.0894,E1 25.1572,E2 460.2269} C_DIS
LIN {X 88.1055,Y -14.3704,Z 93,A -13.8527,B 24.9178,C -2.0935,E1 25.1579,E2 458.8219} C_DIS
LIN {X 88.5732,Y -11.1298,Z 93,A -11.7593,B 24.9173,C -2.0999,E1 25.1587,E2 456.7255} C_DIS
LIN {X 88.8211,Y -8.9383,Z 93,A -10.3604,B 24.917,C -2.1039,E1 25.1591,E2 455.3257} C_DIS
LIN {X 89.0891,Y -5.6752,Z 93,A -8.2726,B 24.9165,C -2.1102,E1 25.1595,E2 453.2355} C_DIS
LIN {X 89.2095,Y -3.3032,Z 93,A -6.7787,B 24.9162,C -2.1139,E1 25.1597,E2 451.7415} C_DIS
LIN {X 89.2678,Y -0.5869,Z 93,A -5.0427,B 24.9158,C -2.1193,E1 25.1597,E2 450.0032} C_DIS
LIN {X 89.2488,Y 1.92,Z 93,A -3.4159,B 24.9153,C -2.1251,E1 25.1597,E2 448.3725} C_DIS
LIN {X 89.1145,Y 5.2606,Z 93,A -1.298,B 24.9148,C -2.1309,E1 25.1594,E2 446.2534} C_DIS
LIN {X 88.9446,Y 7.6205,Z 93,A 0.1882,B 24.9145,C -2.1346,E1 25.1591,E2 444.7674} C_DIS
LIN {X 88.7275,Y 9.8331,Z 93,A 1.6081,B 24.9142,C -2.1388,E1 25.1587,E2 443.3457} C_DIS
LIN {X 88.4579,Y 12.0191,Z 93,A 3.0113,B 24.9139,C -2.1429,E1 25.1582,E2 441.9412} C_DIS
LIN {X 88.1372,Y 14.1809,Z 93,A 4.6305,B 24.9129,C -2.1551,E1 25.1575,E2 440.3028} C_DIS
LIN {X 87.5571,Y 17.407,Z 93,A 6.4944,B 24.9131,C -2.153,E1 25.1565,E2 438.4547} C_DIS
LIN {X 87.1048,Y 19.5446,Z 93,A 7.8884,B 24.9127,C -2.157,E1 25.1557,E2 437.0593} C_DIS
LIN {X 86.5945,Y 21.6946,Z 93,A 9.2962,B 24.9124,C -2.161,E1 25.1548,E2 435.6502} C_DIS
LIN {X 86.0371,Y 23.8092,Z 93,A 10.6915,B 24.9121,C -2.165,E1 25.1537,E2 434.2536} C_DIS
LIN {X 85.483,Y 25.7244,Z 93,A 11.9612,B 24.9118,C -2.1685,E1 25.1527,E2 432.9829} C_DIS
Enddeposition()
END
